{warning 'header is generated please add your documentation'}
METHOD testAnyStringIsEmpty : BOOL
VAR_INPUT
	inputStruct	: isEmptyDataStr;
	testNumber 	: USINT;
END_VAR

VAR
	message : STRING;
END_VAR
THIS^.reset();

IF (inputStruct.typeToTest = TypeToTest.TEST_WSTRING) THEN
	THIS^.assertorContainer.assertor.assert.strings.anyString.isEmpty(
		stringToCheck 	:= inputStruct.WStringToTest,
		message			:= ''
	);
					
ELSIF  (inputStruct.typeToTest = TypeToTest.TEST_STRING ) THEN
	THIS^.assertorContainer.assertor.assert.strings.anyString.isEmpty(
		stringToCheck 	:= inputStruct.StringToTest,
		message			:= ''
	);
	
END_IF

message	:= CONCAT( 'Test Number ', TO_STRING(testNumber));
message	:= CONCAT( message, ' during function AnyString.isEmpty ');
message	:= CONCAT( Message , ' has failed ');

THIS^.AssertEquals_BOOL(
	Expected 	:= inputStruct.expectedResult,
	Actual 		:= THIS^.assertorContainer.wasAssertionWrong,
	Message 	:= message
);
END_METHOD

(*

short summary
=============

.. <legal notes>

legal notes
=================
| SPDX-FileCopyrightText: © 2023 ekvip automation GmbH <info@ekvip.de>
| SPDX-License-Identifier: Apache-2.0
| For details check: Apache-2.0_

.. _Apache-2.0: https://www.apache.org/licenses/LICENSE-2.0

.. </legal notes>

parameters
==========

*)

{warning 'header is generated please add your documentation'}
METHOD testAnyStringIsEqualTo : BOOL
VAR_INPUT
	inputStruct	: isEqualToDataStr;
	testNumber 	: USINT;
END_VAR

VAR
	message : STRING;
END_VAR
THIS^.reset();

IF (inputStruct.typeToTest = TypeToTest.TEST_WSTRING) THEN
	THIS^.assertorContainer.assertor.assert.strings.anyString.isEqualTo(
		stringToCheck 	:= inputStruct.WStringToTest,
		expected		:= inputStruct.EqualToWString,
		ignoreCases     := inputStruct.IgnoreCases,
		message			:= ''	 	
	);
					
ELSIF  (inputStruct.typeToTest = TypeToTest.TEST_STRING ) THEN
	THIS^.assertorContainer.assertor.assert.strings.anyString.isEqualTo(
		stringToCheck 	:= inputStruct.StringToTest,
		expected		:= inputStruct.EqualToString,
		ignoreCases     := inputStruct.IgnoreCases,
		message			:= ''
	);
	
END_IF

message	:= CONCAT( 'Test Number ', TO_STRING(testNumber));
message	:= CONCAT( message, ' during function AnyString.isEqualTo ');
message	:= CONCAT( Message , ' has failed ');

THIS^.AssertEquals_BOOL(
	Expected 	:= inputStruct.expectedResult,
	Actual 		:= THIS^.assertorContainer.wasAssertionWrong,
	Message 	:= message
);
END_METHOD

(*

short summary
=============

.. <legal notes>

legal notes
=================
| SPDX-FileCopyrightText: © 2023 ekvip automation GmbH <info@ekvip.de>
| SPDX-License-Identifier: Apache-2.0
| For details check: Apache-2.0_

.. _Apache-2.0: https://www.apache.org/licenses/LICENSE-2.0

.. </legal notes>

parameters
==========

*)

{warning 'header is generated please add your documentation'}
METHOD testAnyStringIsNotEmpty : BOOL
VAR_INPUT
	inputStruct	: isEmptyDataStr;
	testNumber 	: USINT;
END_VAR

VAR
	message : STRING;
END_VAR
THIS^.reset();

IF (inputStruct.typeToTest = TypeToTest.TEST_WSTRING) THEN
	THIS^.assertorContainer.assertor.assert.strings.anyString.isNotEmpty(
		stringToCheck 	:= inputStruct.WStringToTest,
		message			:= ''
	);
					
ELSIF  (inputStruct.typeToTest = TypeToTest.TEST_STRING ) THEN
	THIS^.assertorContainer.assertor.assert.strings.anyString.isNotEmpty(
		stringToCheck 	:= inputStruct.StringToTest,
		message			:= ''
	);
	
END_IF

message	:= CONCAT( 'Test Number ', TO_STRING(testNumber));
message	:= CONCAT( message, ' during function AnyString.isNotEmpty ');
message	:= CONCAT( Message , ' has failed ');

THIS^.AssertEquals_BOOL(
	Expected 	:= inputStruct.expectedResult,
	Actual 		:= THIS^.assertorContainer.wasAssertionWrong,
	Message 	:= message
);
END_METHOD

(*

short summary
=============

.. <legal notes>

legal notes
=================
| SPDX-FileCopyrightText: © 2023 ekvip automation GmbH <info@ekvip.de>
| SPDX-License-Identifier: Apache-2.0
| For details check: Apache-2.0_

.. _Apache-2.0: https://www.apache.org/licenses/LICENSE-2.0

.. </legal notes>

parameters
==========

*)

{warning 'header is generated please add your documentation'}
METHOD testAnyStringIsNotEqualTo : BOOL
VAR_INPUT
	inputStruct	: isEqualToDataStr;
	testNumber 	: USINT;
END_VAR

VAR
	message : STRING;
END_VAR
THIS^.reset();

IF (inputStruct.typeToTest = TypeToTest.TEST_WSTRING) THEN
	THIS^.assertorContainer.assertor.assert.strings.anyString.isNotEqualTo(
		stringToCheck 	:= inputStruct.WStringToTest,
		unexpected		:= inputStruct.EqualToWString,
		ignoreCases     := inputStruct.IgnoreCases,
		message			:= ''	 	
	);
					
ELSIF  (inputStruct.typeToTest = TypeToTest.TEST_STRING ) THEN
	THIS^.assertorContainer.assertor.assert.strings.anyString.isNotEqualTo(
		stringToCheck 	:= inputStruct.StringToTest,
		unexpected		:= inputStruct.EqualToString,
		ignoreCases     := inputStruct.IgnoreCases,
		message			:= ''
	);
	
END_IF

message	:= CONCAT( 'Test Number ', TO_STRING(testNumber));
message	:= CONCAT( message, ' during function AnyString.isNotEqualTo ');
message	:= CONCAT( Message , ' has failed ');

THIS^.AssertEquals_BOOL(
	Expected 	:= inputStruct.expectedResult,
	Actual 		:= THIS^.assertorContainer.wasAssertionWrong,
	Message 	:= message
);
END_METHOD

(*

short summary
=============

.. <legal notes>

legal notes
=================
| SPDX-FileCopyrightText: © 2023 ekvip automation GmbH <info@ekvip.de>
| SPDX-License-Identifier: Apache-2.0
| For details check: Apache-2.0_

.. _Apache-2.0: https://www.apache.org/licenses/LICENSE-2.0

.. </legal notes>

parameters
==========

*)

{warning 'header is generated please add your documentation'}
METHOD testAnyStringLengthBetween
VAR_INPUT
	inputStruct	: IsLengthBetweenBasicData;
	testNumber	: USINT;
END_VAR

VAR
	message	: STRING;
END_VAR

THIS^.reset();

IF (inputStruct.typeToTest = TypeToTest.TEST_WSTRING) THEN	
	THIS^.assertorContainer.assertor.assert.strings.anyString.lenghtIsBetween( 
		stringToCheck	:=	inputStruct.wstringToTest, 
		maxLenght		:=	inputStruct.maxLength,
		minLenght   	:=  inputStruct.minLength,
		message			:=	''          
	);
				
ELSIF  (inputStruct.typeToTest = TypeToTest.TEST_STRING ) THEN
    THIS^.assertorContainer.assertor.assert.strings.anyString.lenghtIsBetween( 
		stringToCheck	:=	inputStruct.stringToTest, 
		maxLenght		:=	inputStruct.maxLength,
		minLenght   	:=  inputStruct.minLength,
		message			:=	''          
	);
END_IF

message	:= CONCAT( 'Test Number ', TO_STRING(testNumber));
message	:= CONCAT( message, ' during function AnyString.isLengthBetween ');
message	:= CONCAT( Message , ' has failed ');
	
THIS^.AssertEquals_BOOL(
	Expected 	:= inputStruct.expectedResult,
	Actual 		:= THIS^.assertorContainer.wasAssertionWrong,
	Message 	:= message
);
	
//TEST_FINISHED();
END_METHOD

(*

short summary
=============

.. <legal notes>

legal notes
=================
| SPDX-FileCopyrightText: © 2023 ekvip automation GmbH <info@ekvip.de>
| SPDX-License-Identifier: Apache-2.0
| For details check: Apache-2.0_

.. _Apache-2.0: https://www.apache.org/licenses/LICENSE-2.0

.. </legal notes>

parameters
==========

*)

{warning 'header is generated please add your documentation'}
METHOD testAnyStringLengthIs
VAR_INPUT
	inputStruct	:IsLengthBasicData;
	testNumber :USINT;
END_VAR

VAR
	message: STRING;
END_VAR


THIS^.reset();

IF (inputStruct.typeToTest = TypeToTest.TEST_WSTRING) THEN
	IF (inputStruct.funcType = FunctionType.EXACT) THEN 
		THIS^.assertorContainer.assertor.assert.strings.anyString.lenghtIsExact( 
			stringToCheck	:=	inputStruct.wstringToTest, 
			expectedLength	:=	inputStruct.expectedLength,
			message			:=	''          
		);
	ELSIF (inputStruct.funcType = FunctionType.MAXIMUM) THEN
		THIS^.assertorContainer.assertor.assert.strings.anyString.lenghtIsMax( 
			stringToCheck	:=	inputStruct.wstringToTest, 
			maxLength		:=	inputStruct.expectedLength,
			message			:=	''
		);
	ELSIF (inputStruct.funcType = FunctionType.MINIMUM) THEN
		THIS^.assertorContainer.assertor.assert.strings.anyString.lenghtIsMin( 
			stringToCheck	:=	inputStruct.wstringToTest, 
			minLength		:=	inputStruct.expectedLength,
			message			:=	''
		);
	END_IF;
				
ELSIF  (inputStruct.typeToTest = TypeToTest.TEST_STRING ) THEN
    IF (inputStruct.funcType = FunctionType.EXACT) THEN 
		THIS^.assertorContainer.assertor.assert.strings.anyString.lenghtIsExact( 
			stringToCheck	:=	inputStruct.stringToTest, 
			expectedLength	:=	inputStruct.expectedLength,
			message			:=	''         
		);
	ELSIF (inputStruct.funcType = FunctionType.MAXIMUM) THEN
		THIS^.assertorContainer.assertor.assert.strings.anyString.lenghtIsMax( 
			stringToCheck	:=	inputStruct.stringToTest, 
			maxLength		:=	inputStruct.expectedLength,
			message			:=	''        
		);
	ELSIF (inputStruct.funcType = FunctionType.MINIMUM) THEN
		THIS^.assertorContainer.assertor.assert.strings.anyString.lenghtIsMin( 
			stringToCheck	:=	inputStruct.stringToTest, 
			minLength		:=	inputStruct.expectedLength,
			message			:=	''          
		);
	END_IF;

END_IF

message	:= CONCAT( 'Test Number ', TO_STRING(testNumber));
message	:= CONCAT( message, ' during function AnyString.isLength ');
message	:= CONCAT( message , TO_STRING(inputStruct.funcType));
message	:= CONCAT( Message , ' has failed ');
	
THIS^.AssertEquals_BOOL(
	Expected 	:= inputStruct.expectedResult,
	Actual 		:= THIS^.assertorContainer.wasAssertionWrong,
	Message 	:= message
);
	
//TEST_FINISHED();
END_METHOD

(*

short summary
=============

.. <legal notes>

legal notes
=================
| SPDX-FileCopyrightText: © 2023 ekvip automation GmbH <info@ekvip.de>
| SPDX-License-Identifier: Apache-2.0
| For details check: Apache-2.0_

.. _Apache-2.0: https://www.apache.org/licenses/LICENSE-2.0

.. </legal notes>

parameters
==========

*)

{warning 'header is generated please add your documentation'}
METHOD testAnyStringStartsWith : BOOL
VAR_INPUT
	inputStruct	: containsDataStr;
	testNumber 	: USINT;
END_VAR

VAR
	message : STRING;
END_VAR
THIS^.reset();

IF (inputStruct.typeToTest = TypeToTest.TEST_WSTRING) THEN
	THIS^.assertorContainer.assertor.assert.strings.anyString.startsWith(
		stringToCheck	:= inputStruct.WStringToTest,
		start			:= inputStruct.WStringToContain,
		ignoreCases		:= inputStruct.IgnoreCases,
		trim			:= inputStruct.Trim,
		message			:= ''
	);
					
ELSIF  (inputStruct.typeToTest = TypeToTest.TEST_STRING ) THEN
	THIS^.assertorContainer.assertor.assert.strings.anyString.startsWith(
		stringToCheck	:= inputStruct.StringToTest,
		start			:= inputStruct.StringToContain,
		ignoreCases		:= inputStruct.IgnoreCases,
		trim			:= inputStruct.Trim,
		message			:= ''
	);

END_IF

message	:= CONCAT( 'Test Number ', TO_STRING(testNumber));
message	:= CONCAT( message, ' during function AnyString.startsWith ');
message	:= CONCAT( Message , ' has failed ');

THIS^.AssertEquals_BOOL(
	Expected 	:= inputStruct.expectedResult,
	Actual 		:= THIS^.assertorContainer.wasAssertionWrong,
	Message 	:= message
);
END_METHOD

(*

short summary
=============

.. <legal notes>

legal notes
=================
| SPDX-FileCopyrightText: © 2023 ekvip automation GmbH <info@ekvip.de>
| SPDX-License-Identifier: Apache-2.0
| For details check: Apache-2.0_

.. _Apache-2.0: https://www.apache.org/licenses/LICENSE-2.0

.. </legal notes>

parameters
==========

*)

{warning 'header is generated please add your documentation'}
METHOD testAsciiEndsWith : BOOL
VAR_INPUT
	inputStruct	: containsDataStr;
	testNumber 	: USINT;
END_VAR

VAR
	message : STRING;
END_VAR
THIS^.reset();

THIS^.assertorContainer.assertor.assert.strings.ascii.endsWith(
	stringToCheck	:= inputStruct.StringToTest,
	end				:= inputStruct.StringToContain,
	ignoreCases		:= inputStruct.IgnoreCases,
	trim			:= inputStruct.Trim,
	message			:= ''
);


message	:= CONCAT( 'Test Number ', TO_STRING(testNumber));
message	:= CONCAT( message, ' during function Ascii.endsWith ');
message	:= CONCAT( Message , ' has failed ');

THIS^.AssertEquals_BOOL(
	Expected 	:= inputStruct.expectedResult,
	Actual 		:= THIS^.assertorContainer.wasAssertionWrong,
	Message 	:= message
);
END_METHOD

(*

short summary
=============

.. <legal notes>

legal notes
=================
| SPDX-FileCopyrightText: © 2023 ekvip automation GmbH <info@ekvip.de>
| SPDX-License-Identifier: Apache-2.0
| For details check: Apache-2.0_

.. _Apache-2.0: https://www.apache.org/licenses/LICENSE-2.0

.. </legal notes>

parameters
==========

*)

{warning 'header is generated please add your documentation'}
METHOD testAsciiIsEmpty : BOOL
VAR_INPUT
	inputStruct	: isEmptyDataStr;
	testNumber 	: USINT;
END_VAR

VAR
	message : STRING;
END_VAR
THIS^.reset();

THIS^.assertorContainer.assertor.assert.strings.anyString.isEmpty(
	stringToCheck 	:= inputStruct.StringToTest,
	message			:= ''
);

message	:= CONCAT( 'Test Number ', TO_STRING(testNumber));
message	:= CONCAT( message, ' during function Ascii.isEmpty ');
message	:= CONCAT( Message , ' has failed ');

THIS^.AssertEquals_BOOL(
	Expected 	:= inputStruct.expectedResult,
	Actual 		:= THIS^.assertorContainer.wasAssertionWrong,
	Message 	:= message
);
END_METHOD

(*

short summary
=============

.. <legal notes>

legal notes
=================
| SPDX-FileCopyrightText: © 2023 ekvip automation GmbH <info@ekvip.de>
| SPDX-License-Identifier: Apache-2.0
| For details check: Apache-2.0_

.. _Apache-2.0: https://www.apache.org/licenses/LICENSE-2.0

.. </legal notes>

parameters
==========

*)

{warning 'header is generated please add your documentation'}
METHOD testAsciiIsEqualTo : BOOL
VAR_INPUT
	inputStruct	: isEqualToDataStr;
	testNumber 	: USINT;
END_VAR

VAR
	message : STRING;
END_VAR
THIS^.reset();

THIS^.assertorContainer.assertor.assert.strings.ascii.isEqualTo(
	stringToCheck 	:= inputStruct.StringToTest,
	expected		:= inputStruct.EqualToString,
	ignoreCases     := inputStruct.IgnoreCases,
	message			:= ''	 	
);

message	:= CONCAT( 'Test Number ', TO_STRING(testNumber));
message	:= CONCAT( message, ' during function Ascii.isEqualTo ');
message	:= CONCAT( Message , ' has failed ');

THIS^.AssertEquals_BOOL(
	Expected 	:= inputStruct.expectedResult,
	Actual 		:= THIS^.assertorContainer.wasAssertionWrong,
	Message 	:= message
);
END_METHOD

(*

short summary
=============

.. <legal notes>

legal notes
=================
| SPDX-FileCopyrightText: © 2023 ekvip automation GmbH <info@ekvip.de>
| SPDX-License-Identifier: Apache-2.0
| For details check: Apache-2.0_

.. _Apache-2.0: https://www.apache.org/licenses/LICENSE-2.0

.. </legal notes>

parameters
==========

*)

{warning 'header is generated please add your documentation'}
METHOD testAsciiIsNotEmpty : BOOL
VAR_INPUT
	inputStruct	: isEmptyDataStr;
	testNumber 	: USINT;
END_VAR

VAR
	message : STRING;
END_VAR
THIS^.reset();

THIS^.assertorContainer.assertor.assert.strings.anyString.isNotEmpty(
	stringToCheck 	:= inputStruct.StringToTest,
	message			:= ''
);

message	:= CONCAT( 'Test Number ', TO_STRING(testNumber));
message	:= CONCAT( message, ' during function Ascii.isNotEmpty ');
message	:= CONCAT( Message , ' has failed ');

THIS^.AssertEquals_BOOL(
	Expected 	:= inputStruct.expectedResult,
	Actual 		:= THIS^.assertorContainer.wasAssertionWrong,
	Message 	:= message
);
END_METHOD

(*

short summary
=============

.. <legal notes>

legal notes
=================
| SPDX-FileCopyrightText: © 2023 ekvip automation GmbH <info@ekvip.de>
| SPDX-License-Identifier: Apache-2.0
| For details check: Apache-2.0_

.. _Apache-2.0: https://www.apache.org/licenses/LICENSE-2.0

.. </legal notes>

parameters
==========

*)

{warning 'header is generated please add your documentation'}
METHOD testAsciiIsNotEqualTo : BOOL
VAR_INPUT
	inputStruct	: isEqualToDataStr;
	testNumber 	: USINT;
END_VAR

VAR
	message : STRING;
END_VAR
THIS^.reset();

THIS^.assertorContainer.assertor.assert.strings.anyString.isNotEqualTo(
	stringToCheck 	:= inputStruct.StringToTest,
	unexpected		:= inputStruct.EqualToString,
	ignoreCases     := inputStruct.IgnoreCases,
	message			:= ''	 	
);

message	:= CONCAT( 'Test Number ', TO_STRING(testNumber));
message	:= CONCAT( message, ' during function Ascii.isNotEqualTo ');
message	:= CONCAT( Message , ' has failed ');

THIS^.AssertEquals_BOOL(
	Expected 	:= inputStruct.expectedResult,
	Actual 		:= THIS^.assertorContainer.wasAssertionWrong,
	Message 	:= message
);
END_METHOD

(*

short summary
=============

.. <legal notes>

legal notes
=================
| SPDX-FileCopyrightText: © 2023 ekvip automation GmbH <info@ekvip.de>
| SPDX-License-Identifier: Apache-2.0
| For details check: Apache-2.0_

.. _Apache-2.0: https://www.apache.org/licenses/LICENSE-2.0

.. </legal notes>

parameters
==========

*)

{warning 'header is generated please add your documentation'}
METHOD testAsciiStartsWith : BOOL
VAR_INPUT
	inputStruct	: containsDataStr;
	testNumber 	: USINT;
END_VAR

VAR
	message : STRING;
END_VAR
THIS^.reset();

THIS^.assertorContainer.assertor.assert.strings.ascii.startsWith(
	stringToCheck	:= inputStruct.StringToTest,
	start			:= inputStruct.StringToContain,
	ignoreCases		:= inputStruct.IgnoreCases,
	trim			:= inputStruct.Trim,
	message			:= ''
);


message	:= CONCAT( 'Test Number ', TO_STRING(testNumber));
message	:= CONCAT( message, ' during function Ascii.startsWith ');
message	:= CONCAT( Message , ' has failed ');

THIS^.AssertEquals_BOOL(
	Expected 	:= inputStruct.expectedResult,
	Actual 		:= THIS^.assertorContainer.wasAssertionWrong,
	Message 	:= message
);
END_METHOD

(*

short summary
=============

.. <legal notes>

legal notes
=================
| SPDX-FileCopyrightText: © 2023 ekvip automation GmbH <info@ekvip.de>
| SPDX-License-Identifier: Apache-2.0
| For details check: Apache-2.0_

.. _Apache-2.0: https://www.apache.org/licenses/LICENSE-2.0

.. </legal notes>

parameters
==========

*)

{warning 'header is generated please add your documentation'}
METHOD testAsciiStringContains : BOOL
VAR_INPUT
	inputStruct	: containsDataStr;
	testNumber :USINT;
END_VAR

VAR
	message : STRING;
END_VAR
THIS^.reset();

THIS^.assertorContainer.assertor.assert.strings.ascii.contains(
	stringToCheck 	:= inputStruct.StringToTest,
	searchString	:= inputStruct.StringToContain, 
	ignoreCases		:= inputStruct.IgnoreCases,
	message         := ''
);

message	:= CONCAT( 'Test Number ', TO_STRING(testNumber));
message	:= CONCAT( message, ' during function Ascii.contains ');
message	:= CONCAT( Message , ' has failed ');

THIS^.AssertEquals_BOOL(
	Expected 	:= inputStruct.expectedResult,
	Actual 		:= THIS^.assertorContainer.wasAssertionWrong,
	Message 	:= message
);
END_METHOD

(*

short summary
=============

.. <legal notes>

legal notes
=================
| SPDX-FileCopyrightText: © 2023 ekvip automation GmbH <info@ekvip.de>
| SPDX-License-Identifier: Apache-2.0
| For details check: Apache-2.0_

.. _Apache-2.0: https://www.apache.org/licenses/LICENSE-2.0

.. </legal notes>

parameters
==========

*)

{warning 'header is generated please add your documentation'}
METHOD testAsciiStringContainsNo : BOOL
VAR_INPUT
	inputStruct	: containsDataStr;
	testNumber 	: USINT;
END_VAR

VAR
	message : STRING;
END_VAR
THIS^.reset();

THIS^.assertorContainer.assertor.assert.strings.utf16.containsNo(
	stringToCheck 	:= inputStruct.WStringToTest,
	searchString	:= inputStruct.WStringToContain, 
	ignoreCases		:= inputStruct.IgnoreCases,
	message         := ''
);

message	:= CONCAT( 'Test Number ', TO_STRING(testNumber));
message	:= CONCAT( message, ' during function Ascii.containsNo ');
message	:= CONCAT( Message , ' has failed ');

THIS^.AssertEquals_BOOL(
	Expected 	:= inputStruct.expectedResult,
	Actual 		:= THIS^.assertorContainer.wasAssertionWrong,
	Message 	:= message
);
END_METHOD

(*

short summary
=============

.. <legal notes>

legal notes
=================
| SPDX-FileCopyrightText: © 2023 ekvip automation GmbH <info@ekvip.de>
| SPDX-License-Identifier: Apache-2.0
| For details check: Apache-2.0_

.. _Apache-2.0: https://www.apache.org/licenses/LICENSE-2.0

.. </legal notes>

parameters
==========

*)

{warning 'header is generated please add your documentation'}
METHOD testAsciiStringLengthBetween
VAR_INPUT
	inputStruct	: IsLengthBetweenBasicData;
	testNumber 	: USINT;
END_VAR

VAR
	message : STRING;
END_VAR
THIS^.reset();

THIS^.assertorContainer.assertor.assert.strings.ascii.lenghtIsBetween( 
	stringToCheck	:=	inputStruct.stringToTest, 
	maxLenght		:=	inputStruct.maxLength,
	minLenght   	:=  inputStruct.minLength,
	message			:=	''          
);


message	:= CONCAT( 'Test Number ', TO_STRING(testNumber));
message	:= CONCAT( message, ' during function Ascii.isLengthBetween ');
message	:= CONCAT( Message , ' has failed ');
	
THIS^.AssertEquals_BOOL(
	Expected 	:= inputStruct.expectedResult,
	Actual 		:= THIS^.assertorContainer.wasAssertionWrong,
	Message 	:= message
);
END_METHOD

(*

short summary
=============

.. <legal notes>

legal notes
=================
| SPDX-FileCopyrightText: © 2023 ekvip automation GmbH <info@ekvip.de>
| SPDX-License-Identifier: Apache-2.0
| For details check: Apache-2.0_

.. _Apache-2.0: https://www.apache.org/licenses/LICENSE-2.0

.. </legal notes>

parameters
==========

*)

{warning 'header is generated please add your documentation'}
METHOD testAsciiStringlengthIs
VAR_INPUT
	inputStruct	:IsLengthBasicData;
	testNumber :USINT;
END_VAR

VAR
	message: STRING;
END_VAR

THIS^.reset();

IF (inputStruct.funcType = FunctionType.EXACT) THEN 
	THIS^.assertorContainer.assertor.assert.strings.ascii.lenghtIsExact( 
		stringToCheck	:=	inputStruct.stringToTest, 
		expectedLength	:=	TO_USINT(inputStruct.expectedLength),
		message			:=	''          
	);
ELSIF (inputStruct.funcType = FunctionType.MAXIMUM) THEN
	THIS^.assertorContainer.assertor.assert.strings.ascii.lenghtIsMax( 
		stringToCheck	:=	inputStruct.stringToTest, 
		maxLength		:=	TO_USINT(inputStruct.expectedLength),
		message			:=	''         
	);
ELSIF (inputStruct.funcType = FunctionType.MINIMUM) THEN
	THIS^.assertorContainer.assertor.assert.strings.ascii.lenghtIsMin( 
		stringToCheck	:=	inputStruct.stringToTest, 
		minLength		:=	TO_USINT(inputStruct.expectedLength),
		message			:=	''          
	);
END_IF;

message	:= CONCAT( 'Test Number ', TO_STRING(testNumber));
message	:= CONCAT( message, ' during function AsciiString.isLength ');
message	:= CONCAT( message , TO_STRING(inputStruct.funcType));
message	:= CONCAT( Message , ' has failed ');

THIS^.AssertEquals_BOOL(
	Expected 	:= inputStruct.expectedResult,
	Actual 		:= THIS^.assertorContainer.wasAssertionWrong,
	Message		:= message
);
END_METHOD

(*

short summary
=============

.. <legal notes>

legal notes
=================
| SPDX-FileCopyrightText: © 2023 ekvip automation GmbH <info@ekvip.de>
| SPDX-License-Identifier: Apache-2.0
| For details check: Apache-2.0_

.. _Apache-2.0: https://www.apache.org/licenses/LICENSE-2.0

.. </legal notes>

parameters
==========

*)

{warning 'header is generated please add your documentation'}
METHOD testUtf16EndsWith : BOOL
VAR_INPUT
	inputStruct	: containsDataStr;
	testNumber 	: USINT;
END_VAR

VAR
	message : STRING;
END_VAR
THIS^.reset();

THIS^.assertorContainer.assertor.assert.strings.utf16.endsWith(
	stringToCheck	:= inputStruct.WStringToTest,
	end				:= inputStruct.WStringToContain,
	ignoreCases		:= inputStruct.IgnoreCases,
	trim			:= inputStruct.Trim,
	message			:= ''
);

message	:= CONCAT( 'Test Number ', TO_STRING(testNumber));
message	:= CONCAT( message, ' during function UTF16.endsWith ');
message	:= CONCAT( Message , ' has failed ');

THIS^.AssertEquals_BOOL(
	Expected 	:= inputStruct.expectedResult,
	Actual 		:= THIS^.assertorContainer.wasAssertionWrong,
	Message 	:= message
);
END_METHOD

(*

short summary
=============

.. <legal notes>

legal notes
=================
| SPDX-FileCopyrightText: © 2023 ekvip automation GmbH <info@ekvip.de>
| SPDX-License-Identifier: Apache-2.0
| For details check: Apache-2.0_

.. _Apache-2.0: https://www.apache.org/licenses/LICENSE-2.0

.. </legal notes>

parameters
==========

*)

{warning 'header is generated please add your documentation'}
METHOD testUtf16IsEmpty : BOOL
VAR_INPUT
	inputStruct	: isEmptyDataStr;
	testNumber 	: USINT;
END_VAR

VAR
	message : STRING;
END_VAR
THIS^.reset();

THIS^.assertorContainer.assertor.assert.strings.anyString.isEmpty(
	stringToCheck 	:= inputStruct.WStringToTest,
	message			:= ''
);

message	:= CONCAT( 'Test Number ', TO_STRING(testNumber));
message	:= CONCAT( message, ' during function UTF16.isEmpty ');
message	:= CONCAT( Message , ' has failed ');

THIS^.AssertEquals_BOOL(
	Expected 	:= inputStruct.expectedResult,
	Actual 		:= THIS^.assertorContainer.wasAssertionWrong,
	Message 	:= message
);
END_METHOD

(*

short summary
=============

.. <legal notes>

legal notes
=================
| SPDX-FileCopyrightText: © 2023 ekvip automation GmbH <info@ekvip.de>
| SPDX-License-Identifier: Apache-2.0
| For details check: Apache-2.0_

.. _Apache-2.0: https://www.apache.org/licenses/LICENSE-2.0

.. </legal notes>

parameters
==========

*)

{warning 'header is generated please add your documentation'}
METHOD testUtf16IsEqualTo : BOOL
VAR_INPUT
	inputStruct	: isEqualToDataStr;
	testNumber 	: USINT;
END_VAR

VAR
	message : STRING;
END_VAR
THIS^.reset();

THIS^.assertorContainer.assertor.assert.strings.anyString.isEqualTo(
	stringToCheck 	:= inputStruct.WStringToTest,
	expected		:= inputStruct.EqualToWString,
	ignoreCases     := inputStruct.IgnoreCases,
	message			:= ''	 	
);
   
message	:= CONCAT( 'Test Number ', TO_STRING(testNumber));
message	:= CONCAT( message, ' during function UTF16.isEqualTo ');
message	:= CONCAT( Message , ' has failed ');

THIS^.AssertEquals_BOOL(
	Expected 	:= inputStruct.expectedResult,
	Actual 		:= THIS^.assertorContainer.wasAssertionWrong,
	Message 	:= message
);
END_METHOD

(*

short summary
=============

.. <legal notes>

legal notes
=================
| SPDX-FileCopyrightText: © 2023 ekvip automation GmbH <info@ekvip.de>
| SPDX-License-Identifier: Apache-2.0
| For details check: Apache-2.0_

.. _Apache-2.0: https://www.apache.org/licenses/LICENSE-2.0

.. </legal notes>

parameters
==========

*)

{warning 'header is generated please add your documentation'}
METHOD testUtf16IsNotEmpty : BOOL
VAR_INPUT
	inputStruct	: isEmptyDataStr;
	testNumber 	: USINT;
END_VAR

VAR
	message : STRING;
END_VAR
THIS^.reset();

THIS^.assertorContainer.assertor.assert.strings.anyString.isNotEmpty(
	stringToCheck 	:= inputStruct.WStringToTest,
	message			:= ''
);

message	:= CONCAT( 'Test Number ', TO_STRING(testNumber));
message	:= CONCAT( message, ' during function UTF16.isNotEmpty ');
message	:= CONCAT( Message , ' has failed ');

THIS^.AssertEquals_BOOL(
	Expected 	:= inputStruct.expectedResult,
	Actual 		:= THIS^.assertorContainer.wasAssertionWrong,
	Message 	:= message
);
END_METHOD

(*

short summary
=============

.. <legal notes>

legal notes
=================
| SPDX-FileCopyrightText: © 2023 ekvip automation GmbH <info@ekvip.de>
| SPDX-License-Identifier: Apache-2.0
| For details check: Apache-2.0_

.. _Apache-2.0: https://www.apache.org/licenses/LICENSE-2.0

.. </legal notes>

parameters
==========

*)

{warning 'header is generated please add your documentation'}
METHOD testUtf16IsNotEqualTo : BOOL
VAR_INPUT
	inputStruct	: isEqualToDataStr;
	testNumber 	: USINT;
END_VAR

VAR
	message : STRING;
END_VAR
THIS^.reset();

THIS^.assertorContainer.assertor.assert.strings.anyString.isNotEqualTo(
	stringToCheck 	:= inputStruct.WStringToTest,
	unexpected		:= inputStruct.EqualToWString,
	ignoreCases     := inputStruct.IgnoreCases,
	message			:= ''	 	
);
   
message	:= CONCAT( 'Test Number ', TO_STRING(testNumber));
message	:= CONCAT( message, ' during function UTF16.isNotEqualTo ');
message	:= CONCAT( Message , ' has failed ');

THIS^.AssertEquals_BOOL(
	Expected 	:= inputStruct.expectedResult,
	Actual 		:= THIS^.assertorContainer.wasAssertionWrong,
	Message 	:= message
);
END_METHOD

(*

short summary
=============

.. <legal notes>

legal notes
=================
| SPDX-FileCopyrightText: © 2023 ekvip automation GmbH <info@ekvip.de>
| SPDX-License-Identifier: Apache-2.0
| For details check: Apache-2.0_

.. _Apache-2.0: https://www.apache.org/licenses/LICENSE-2.0

.. </legal notes>

parameters
==========

*)

{warning 'header is generated please add your documentation'}
METHOD testUtf16StartsWith : BOOL
VAR_INPUT
	inputStruct	: containsDataStr;
	testNumber 	: USINT;
END_VAR

VAR
	message : STRING;
END_VAR
THIS^.reset();

THIS^.assertorContainer.assertor.assert.strings.utf16.startsWith(
	stringToCheck	:= inputStruct.WStringToTest,
	start			:= inputStruct.WStringToContain,
	ignoreCases		:= inputStruct.IgnoreCases,
	trim			:= inputStruct.Trim,
	message			:= ''
);

message	:= CONCAT( 'Test Number ', TO_STRING(testNumber));
message	:= CONCAT( message, ' during function UTF16.startsWith ');
message	:= CONCAT( Message , ' has failed ');

THIS^.AssertEquals_BOOL(
	Expected 	:= inputStruct.expectedResult,
	Actual 		:= THIS^.assertorContainer.wasAssertionWrong,
	Message 	:= message
);
END_METHOD

(*

short summary
=============

.. <legal notes>

legal notes
=================
| SPDX-FileCopyrightText: © 2023 ekvip automation GmbH <info@ekvip.de>
| SPDX-License-Identifier: Apache-2.0
| For details check: Apache-2.0_

.. _Apache-2.0: https://www.apache.org/licenses/LICENSE-2.0

.. </legal notes>

parameters
==========

*)

{warning 'header is generated please add your documentation'}
METHOD testUtf16StringContains : BOOL
VAR_INPUT
	inputStruct	: containsDataStr;
	testNumber :USINT;
END_VAR

VAR
	message : STRING;
END_VAR
THIS^.reset();

THIS^.assertorContainer.assertor.assert.strings.utf16.contains(
	stringToCheck 	:= inputStruct.WStringToTest,
	searchString	:= inputStruct.WStringToContain, 
	ignoreCases		:= inputStruct.IgnoreCases,
	message         := ''
);

message	:= CONCAT( 'Test Number ', TO_STRING(testNumber));
message	:= CONCAT( message, ' during function UTF16.contains ');
message	:= CONCAT( Message , ' has failed ');

THIS^.AssertEquals_BOOL(
	Expected 	:= inputStruct.expectedResult,
	Actual 		:= THIS^.assertorContainer.wasAssertionWrong,
	Message 	:= message
);
END_METHOD

(*

short summary
=============

.. <legal notes>

legal notes
=================
| SPDX-FileCopyrightText: © 2023 ekvip automation GmbH <info@ekvip.de>
| SPDX-License-Identifier: Apache-2.0
| For details check: Apache-2.0_

.. _Apache-2.0: https://www.apache.org/licenses/LICENSE-2.0

.. </legal notes>

parameters
==========

*)

{warning 'header is generated please add your documentation'}
METHOD testUtf16StringContainsNo : BOOL
VAR_INPUT
	inputStruct	: containsDataStr;
	testNumber 	: USINT;
END_VAR

VAR
	message : STRING;
END_VAR
THIS^.reset();

THIS^.assertorContainer.assertor.assert.strings.utf16.containsNo(
	stringToCheck 	:= inputStruct.WStringToTest,
	searchString	:= inputStruct.WStringToContain, 
	ignoreCases		:= inputStruct.IgnoreCases,
	message         := ''
);

message	:= CONCAT( 'Test Number ', TO_STRING(testNumber));
message	:= CONCAT( message, ' during function UTF16.containsNo ');
message	:= CONCAT( Message , ' has failed ');

THIS^.AssertEquals_BOOL(
	Expected 	:= inputStruct.expectedResult,
	Actual 		:= THIS^.assertorContainer.wasAssertionWrong,
	Message 	:= message
);
END_METHOD

(*

short summary
=============

.. <legal notes>

legal notes
=================
| SPDX-FileCopyrightText: © 2023 ekvip automation GmbH <info@ekvip.de>
| SPDX-License-Identifier: Apache-2.0
| For details check: Apache-2.0_

.. _Apache-2.0: https://www.apache.org/licenses/LICENSE-2.0

.. </legal notes>

parameters
==========

*)

{warning 'header is generated please add your documentation'}
METHOD testUtf16StringLengthBetween
VAR_INPUT
	inputStruct : IsLengthBetweenBasicData;
	testNumber	: USINT;
END_VAR

VAR
	message: STRING;
END_VAR
THIS^.reset();

THIS^.assertorContainer.assertor.assert.strings.utf16.lenghtIsBetween( 
	stringToCheck	:=	inputStruct.wstringToTest, 
	maxLenght		:=	inputStruct.maxLength,
	minLenght   	:=  inputStruct.minLength,
	message			:=	''          
);


message	:= CONCAT( 'Test Number ', TO_STRING(testNumber));
message	:= CONCAT( message, ' during function UTF16.isLengthBetween ');
message	:= CONCAT( Message , ' has failed ');
	
THIS^.AssertEquals_BOOL(
	Expected 	:= inputStruct.expectedResult,
	Actual 		:= THIS^.assertorContainer.wasAssertionWrong,
	Message 	:= message
);
END_METHOD

(*

short summary
=============

.. <legal notes>

legal notes
=================
| SPDX-FileCopyrightText: © 2023 ekvip automation GmbH <info@ekvip.de>
| SPDX-License-Identifier: Apache-2.0
| For details check: Apache-2.0_

.. _Apache-2.0: https://www.apache.org/licenses/LICENSE-2.0

.. </legal notes>

parameters
==========

*)

{warning 'header is generated please add your documentation'}
METHOD testUtf16StringlengthIs
VAR_INPUT
	inputStruct	:IsLengthBasicData;
	testNumber :USINT;
END_VAR

VAR
	message: STRING;
END_VAR

THIS^.reset();

IF (inputStruct.funcType = FunctionType.EXACT) THEN
	THIS^.assertorContainer.assertor.assert.strings.utf16.lenghtIsExact( 
		stringToCheck	:=	inputStruct.wstringToTest, 
		expectedLength	:=	TO_USINT(inputStruct.expectedLength),
		message			:=	''          
	);
ELSIF (inputStruct.funcType = FunctionType.MAXIMUM) THEN
	THIS^.assertorContainer.assertor.assert.strings.utf16.lenghtIsMax( 
		stringToCheck	:=	inputStruct.wstringToTest, 
		maxLength		:=	TO_USINT(inputStruct.expectedLength),
		message			:=	''         
	);
ELSIF (inputStruct.funcType = FunctionType.MINIMUM) THEN
	THIS^.assertorContainer.assertor.assert.strings.utf16.lenghtIsMin( 
		stringToCheck	:=	inputStruct.wstringToTest, 
		minLength		:=	TO_USINT(inputStruct.expectedLength),
		message			:=	' '         
	);
END_IF;

message	:= CONCAT( ' Test Number ', TO_STRING(testNumber));
message	:= CONCAT( message, ' during function UFT16String.isLength ');
message	:= CONCAT( message , TO_STRING(inputStruct.funcType));
message	:= CONCAT( Message , ' has failed ');
	
THIS^.AssertEquals_BOOL(
	Expected 	:= inputStruct.expectedResult,
	Actual 		:= THIS^.assertorContainer.wasAssertionWrong,
	Message 	:= message
);
END_METHOD

END_FUNCTION_BLOCK

// ---- AssertionTester/AssertionTests/TimeAssertions/TimeAssertionsTests.TcPOU
(*

short summary
=============

.. <legal notes>

legal notes
=================
| SPDX-FileCopyrightText: © 2023 ekvip automation GmbH <info@ekvip.de>
| SPDX-License-Identifier: Apache-2.0
| For details check: Apache-2.0_

.. _Apache-2.0: https://www.apache.org/licenses/LICENSE-2.0

.. </legal notes>

methods and properties
======================

*)

{warning 'header is generated please add your documentation'}
FUNCTION_BLOCK TimeAssertionsTests EXTENDS AbstractAssertorTest
VAR CONSTANT
	NUMBER_OF_SETS :INT := 9;
END_VAR
VAR
	simpleTimeValuesToCurrent 	:ARRAY [0..NUMBER_OF_SETS] OF TIME;
	simpleTimeValuesToExpected 	:ARRAY [0..NUMBER_OF_SETS] OF TIME;
	longTimeValuesToCurrent 	:ARRAY [0..NUMBER_OF_SETS] OF LTIME;
	longTimeValuesToExpected 	:ARRAY [0..NUMBER_OF_SETS] OF LTIME;								
END_VAR


assignTimes();

(* Simple time tests *)

THIS^.testSimpleValueIsEqualTo(simpleTimeValuesToCurrent, simpleTimeValuesToExpected);

THIS^.testSimpleValueIsNotEqualTo(simpleTimeValuesToCurrent, mirrorSimpleTimeArray(simpleTimeValuesToExpected));

THIS^.testSimpleValueIsGreaterThan(simpleTimeValuesToCurrent, simpleTimeValuesToExpected);

THIS^.testSimpleValueIsLessThan(simpleTimeValuesToCurrent, simpleTimeValuesToExpected);

THIS^.testSimpleValueIsInRangeOf(simpleTimeValuesToCurrent, simpleTimeValuesToExpected, mirrorSimpleTimeArray(simpleTimeValuesToExpected));

THIS^.testSimpleValueIsMax(simpleTimeValuesToCurrent, mirrorSimpleTimeArray(simpleTimeValuesToExpected));

THIS^.testSimpleValueIsMin(simpleTimeValuesToCurrent, mirrorSimpleTimeArray(simpleTimeValuesToExpected));

THIS^.testSimpleTimeHasExpired(simpleTimeValuesToCurrent, mirrorSimpleTimeArray(simpleTimeValuesToExpected));

THIS^.testSimpleTimeHasNotExpired(simpleTimeValuesToCurrent, mirrorSimpleTimeArray(simpleTimeValuesToExpected));

(* Long time tests *)

THIS^.testLongValueIsEqualTo(longTimeValuesToCurrent, longTimeValuesToExpected);

THIS^.testLongValueIsNotEqualTo(longTimeValuesToCurrent, mirrorLongTimeArray(longTimeValuesToExpected));

THIS^.testLongValueIsGreaterThan(longTimeValuesToCurrent, longTimeValuesToExpected);

THIS^.testLongValueIsLessThan(longTimeValuesToCurrent, longTimeValuesToExpected);

THIS^.testLongValueIsInRangeOf(longTimeValuesToCurrent, longTimeValuesToExpected, mirrorLongTimeArray(longTimeValuesToExpected));

THIS^.testLongValueIsMax(longTimeValuesToCurrent, mirrorLongTimeArray(longTimeValuesToExpected));

THIS^.testLongValueIsMin(longTimeValuesToCurrent, mirrorLongTimeArray(longTimeValuesToExpected));

THIS^.testLongTimeHasExpired(longTimeValuesToCurrent, mirrorlongTimeArray(longTimeValuesToExpected));

THIS^.testLongTimeHasNotExpired(longTimeValuesToCurrent, mirrorlongTimeArray(longTimeValuesToExpected));

(*

short summary
=============

.. <legal notes>

legal notes
=================
| SPDX-FileCopyrightText: © 2023 ekvip automation GmbH <info@ekvip.de>
| SPDX-License-Identifier: Apache-2.0
| For details check: Apache-2.0_

.. _Apache-2.0: https://www.apache.org/licenses/LICENSE-2.0

.. </legal notes>

parameters
==========

*)

{warning 'header is generated please add your documentation'}
METHOD assignTimes
		
// simple time
simpleTimeValuesToCurrent[0] := TIME#0M;					simpleTimeValuesToExpected[0] := TIME#0S;
simpleTimeValuesToCurrent[1] := TIME#0.01667M;				simpleTimeValuesToExpected[1] := TIME#1S;
simpleTimeValuesToCurrent[2] := TIME#1M;					simpleTimeValuesToExpected[2] := TIME#60S;
simpleTimeValuesToCurrent[3] := TIME#60M;					simpleTimeValuesToExpected[3] := TIME#3_600S;
simpleTimeValuesToCurrent[4] := TIME#1440M;					simpleTimeValuesToExpected[4] := TIME#86_400S;
simpleTimeValuesToCurrent[5] := TIME#10_080M;				simpleTimeValuesToExpected[5] := TIME#604_800S;
simpleTimeValuesToCurrent[6] := TIME#20_160M;				simpleTimeValuesToExpected[6] := TIME#1_209_600S;
simpleTimeValuesToCurrent[7] := TIME#40_320M;				simpleTimeValuesToExpected[7] := TIME#2_419_200S;
simpleTimeValuesToCurrent[8] := TIME#60_480M;				simpleTimeValuesToExpected[8] := TIME#3_628_800S;
simpleTimeValuesToCurrent[9] := TIME#4294967295MS;			simpleTimeValuesToExpected[9] := TIME#4294967295MS;

// long time
longTimeValuesToCurrent[0] := LTIME#0MS;					longTimeValuesToExpected[0] := LTIME#0NS;
longTimeValuesToCurrent[1] := LTIME#1_000MS;				longTimeValuesToExpected[1] := LTIME#1000_000_000NS;
longTimeValuesToCurrent[2] := LTIME#60_000MS;				longTimeValuesToExpected[2] := LTIME#60_000_000_000NS;
longTimeValuesToCurrent[3] := LTIME#3_600_000MS;			longTimeValuesToExpected[3] := LTIME#3_600_000_000_000NS;
longTimeValuesToCurrent[4] := LTIME#86_400_000MS;			longTimeValuesToExpected[4] := LTIME#86_400_000_000_000NS;
longTimeValuesToCurrent[5] := LTIME#604_800_000MS;			longTimeValuesToExpected[5] := LTIME#604_800_000_000_000NS;
longTimeValuesToCurrent[6] := LTIME#1_209_600_000MS;		longTimeValuesToExpected[6] := LTIME#1_209_600_000_000_000NS;
longTimeValuesToCurrent[7] := LTIME#2_419_200_000MS;		longTimeValuesToExpected[7] := LTIME#2_419_200_000_000_000NS;
longTimeValuesToCurrent[8] := LTIME#31_557_600_000MS;		longTimeValuesToExpected[8] := LTIME#31_557_600_000_000_000NS;
longTimeValuesToCurrent[9] := LTIME#31_557_600_000MS;		longTimeValuesToExpected[9] := LTIME#213503D23H34M33S709MS551US615NS;
END_METHOD

(*

short summary
=============

.. <legal notes>

legal notes
=================
| SPDX-FileCopyrightText: © 2023 ekvip automation GmbH <info@ekvip.de>
| SPDX-License-Identifier: Apache-2.0
| For details check: Apache-2.0_

.. _Apache-2.0: https://www.apache.org/licenses/LICENSE-2.0

.. </legal notes>

parameters
==========

*)

{warning 'header is generated please add your documentation'}

METHOD mirrorLongTimeArray :ARRAY [0..NUMBER_OF_SETS] OF LTIME
VAR_INPUT
	inputArray :ARRAY [0..NUMBER_OF_SETS] OF LTIME;
END_VAR
VAR
	tempArray :ARRAY [0..NUMBER_OF_SETS] OF LTIME;
	temp :LTIME;
	i :INT;
END_VAR
tempArray := inputArray;

FOR i := 0 TO (NUMBER_OF_SETS/2 - 1) DO
	temp := inputArray[i];
	tempArray[i] := inputArray[NUMBER_OF_SETS - i];
	tempArray[NUMBER_OF_SETS - i] := temp;
END_FOR

mirrorLongTimeArray := tempArray;
END_METHOD

(*

short summary
=============

.. <legal notes>

legal notes
=================
| SPDX-FileCopyrightText: © 2023 ekvip automation GmbH <info@ekvip.de>
| SPDX-License-Identifier: Apache-2.0
| For details check: Apache-2.0_

.. _Apache-2.0: https://www.apache.org/licenses/LICENSE-2.0

.. </legal notes>

parameters
==========

*)

{warning 'header is generated please add your documentation'}

METHOD mirrorSimpleTimeArray :ARRAY [0..NUMBER_OF_SETS] OF TIME
VAR_INPUT
	inputArray :ARRAY [0..NUMBER_OF_SETS] OF TIME;
END_VAR
VAR
	tempArray :ARRAY [0..NUMBER_OF_SETS] OF TIME;
	temp :TIME;
	i :INT;
END_VAR
tempArray := inputArray;

FOR i := 0 TO (NUMBER_OF_SETS/2 - 1) DO
	temp := inputArray[i];
	tempArray[i] := inputArray[NUMBER_OF_SETS - i];
	tempArray[NUMBER_OF_SETS - i] := temp;
END_FOR

mirrorSimpleTimeArray := tempArray;
END_METHOD

(*

short summary
=============

.. <legal notes>

legal notes
=================
| SPDX-FileCopyrightText: © 2023 ekvip automation GmbH <info@ekvip.de>
| SPDX-License-Identifier: Apache-2.0
| For details check: Apache-2.0_

.. _Apache-2.0: https://www.apache.org/licenses/LICENSE-2.0

.. </legal notes>

parameters
==========

*)

{warning 'header is generated please add your documentation'}

METHOD testLongTimeHasExpired
VAR_INPUT
	currentValue :ARRAY [0..NUMBER_OF_SETS] OF LTIME;
	expectedValue :ARRAY [0..NUMBER_OF_SETS] OF LTIME;
END_VAR
VAR
	i :INT;
	message :Tc2_System.T_MaxString;
	timeStamp :LTIME;
	currentTime :LTIME;
	timeout :LTIME;
	timeExpired :BOOL;
END_VAR
VAR CONSTANT
	MAX_TIME :LTIME := TO_LTIME(16#FF_FF_FF_FF_FF_FF_FF_FF);
END_VAR

TEST('TEST--TimeAssertion--testLongTimeHasExpired');

FOR i := 0 TO 9 BY 1 DO
	
	THIS^.assertorContainer.resetAssertor();
	currentTime := LTIME();	
	timeStamp := SEL(currentTime > currentValue[i], currentTime - currentValue[i], currentTime);

	timeExpired := (TO_LINT(timeStamp)) >= (TO_LINT(currentTime));
	THIS^.assertorContainer.assertor.assert.times.long.timeHasExpired(
		timestamp := timeStamp,
		expiringTime := expectedValue[i],
		message := ''
	);
	
	
	
	message := 'TimeAssertionTests';
	message := Tc2_Standard.CONCAT(message, ' -> ');
	message := Tc2_Standard.CONCAT(message, 'longTimeHasExpired');
	message := Tc2_Standard.CONCAT(message, ' -> ');
	message := Tc2_Standard.CONCAT(message, ' Test ');
	message := Tc2_Standard.CONCAT(message, TO_STRING(i));
	message := Tc2_Standard.CONCAT(message, ' -> ');
	message := Tc2_Standard.CONCAT(message, ' currentValue = ');
	message := Tc2_Standard.CONCAT(message, TO_STRING(TO_LINT(currentValue[i])));	
	message := Tc2_Standard.CONCAT(message, ' -> ');
	message := Tc2_Standard.CONCAT(message, ' expectedValue = ');
	message := Tc2_Standard.CONCAT(message, TO_STRING(TO_LINT(expectedValue[i])));
	message := Tc2_Standard.CONCAT(message, ' -> ');
	message := Tc2_Standard.CONCAT(message, ' timestamp = ');
	message := Tc2_Standard.CONCAT(message, TO_STRING(TO_LINT(timeStamp)));
	message := Tc2_Standard.CONCAT(message, ' -> ');
	message := Tc2_Standard.CONCAT(message, ' currentTime = ');
	message := Tc2_Standard.CONCAT(message, TO_STRING(TO_LINT(currentTime)));
	message := Tc2_Standard.CONCAT(message, ' -> ');
	message := Tc2_Standard.CONCAT(message, ' timeExpired = ');
	message := Tc2_Standard.CONCAT(message, TO_STRING(TO_LINT(timeExpired)));
	message := Tc2_Standard.CONCAT(message, ' => ');
	message := Tc2_Standard.CONCAT(message, ' assertionWasWrong = ');
	message := Tc2_Standard.CONCAT(message, TO_STRING(THIS^.assertorContainer.wasAssertionWrong));



	IF (timeExpired) THEN
		THIS^.AssertFALSE(
			Condition := THIS^.assertorContainer.wasAssertionWrong,
			Message := message
		);
	ELSE
		THIS^.AssertTrue(
			Condition := THIS^.assertorContainer.wasAssertionWrong,
			Message := message
		);		
	END_IF
	
END_FOR;


TEST_FINISHED();
END_METHOD

(*

short summary
=============

.. <legal notes>

legal notes
=================
| SPDX-FileCopyrightText: © 2023 ekvip automation GmbH <info@ekvip.de>
| SPDX-License-Identifier: Apache-2.0
| For details check: Apache-2.0_

.. _Apache-2.0: https://www.apache.org/licenses/LICENSE-2.0

.. </legal notes>

parameters
==========

*)

{warning 'header is generated please add your documentation'}

METHOD testLongTimeHasNotExpired
VAR_INPUT
	currentValue :ARRAY [0..NUMBER_OF_SETS] OF LTIME;
	expectedValue :ARRAY [0..NUMBER_OF_SETS] OF LTIME;
END_VAR
VAR
	i :INT;
	message :Tc2_System.T_MaxString;
	 timeStamp :LTIME;
	 currentTime :LTIME;
	 timeout :LTIME;
	 timeExpired :BOOL;
END_VAR
VAR CONSTANT
	MAX_TIME :LTIME := TO_LTIME(16#FF_FF_FF_FF_FF_FF_FF_FF);
END_VAR

TEST('TEST--TimeAssertion--testLongTimeHasNotExpired');

FOR i := 0 TO 9 BY 1 DO
	
	THIS^.assertorContainer.resetAssertor();
	currentTime := LTIME();	
//	timeStamp := SEL(currentTime < currentValue[i], currentTime - currentValue[i], MAX_TIME - currentValue[i] + currentTime);
	timeStamp := SEL(currentTime > currentValue[i], currentTime - currentValue[i], currentTime);

	timeExpired := (TO_LINT(timeStamp)) >= (TO_LINT(currentTime));
	THIS^.assertorContainer.assertor.assert.times.long.timeHasNotExpired(
		timestamp := timeStamp,
		expiringTime := expectedValue[i],
		message := ''
	);
	
	
	
	message := 'TimeAssertionTests';
	message := Tc2_Standard.CONCAT(message, ' -> ');
	message := Tc2_Standard.CONCAT(message, 'longTimeHasNotExpired');
	message := Tc2_Standard.CONCAT(message, ' -> ');
	message := Tc2_Standard.CONCAT(message, ' Test ');
	message := Tc2_Standard.CONCAT(message, TO_STRING(i));
	message := Tc2_Standard.CONCAT(message, ' -> ');
	message := Tc2_Standard.CONCAT(message, ' currentValue = ');
	message := Tc2_Standard.CONCAT(message, TO_STRING(TO_LINT(currentValue[i])));	
	message := Tc2_Standard.CONCAT(message, ' -> ');
	message := Tc2_Standard.CONCAT(message, ' expectedValue = ');
	message := Tc2_Standard.CONCAT(message, TO_STRING(TO_LINT(expectedValue[i])));
	message := Tc2_Standard.CONCAT(message, ' -> ');
	message := Tc2_Standard.CONCAT(message, ' timestamp = ');
	message := Tc2_Standard.CONCAT(message, TO_STRING(TO_LINT(timeStamp)));
	message := Tc2_Standard.CONCAT(message, ' -> ');
	message := Tc2_Standard.CONCAT(message, ' currentTime = ');
	message := Tc2_Standard.CONCAT(message, TO_STRING(TO_LINT(currentTime)));
	message := Tc2_Standard.CONCAT(message, ' -> ');
	message := Tc2_Standard.CONCAT(message, ' timeExpired = ');
	message := Tc2_Standard.CONCAT(message, TO_STRING(TO_LINT(timeExpired)));
	message := Tc2_Standard.CONCAT(message, ' => ');
	message := Tc2_Standard.CONCAT(message, ' assertionWasWrong = ');
	message := Tc2_Standard.CONCAT(message, TO_STRING(THIS^.assertorContainer.wasAssertionWrong));


	IF (NOT timeExpired) THEN
		THIS^.AssertFALSE(
			Condition := THIS^.assertorContainer.wasAssertionWrong,
			Message := message
		);
	ELSE
		THIS^.AssertTrue(
			Condition := THIS^.assertorContainer.wasAssertionWrong,
			Message := message
		);		
	END_IF
	
END_FOR;


TEST_FINISHED();
END_METHOD

(*

short summary
=============

.. <legal notes>

legal notes
=================
| SPDX-FileCopyrightText: © 2023 ekvip automation GmbH <info@ekvip.de>
| SPDX-License-Identifier: Apache-2.0
| For details check: Apache-2.0_

.. _Apache-2.0: https://www.apache.org/licenses/LICENSE-2.0

.. </legal notes>

parameters
==========

*)

{warning 'header is generated please add your documentation'}

METHOD testLongValueIsEqualTo
VAR_INPUT
	currentValue :ARRAY [0..NUMBER_OF_SETS] OF LTIME;
	expectedValue :ARRAY [0..NUMBER_OF_SETS] OF LTIME;
END_VAR
VAR
	i :INT;
	message :Tc2_System.T_MaxString;
END_VAR
TEST('TEST--TimeAssertion--testLongValueIsEqualTo');

FOR i := 0 TO 9 BY 1 DO
	
	THIS^.assertorContainer.resetAssertor();
	THIS^.assertorContainer.assertor.assert.times.long.valueIsEqualTo(
		currentValue := currentValue[i],
		expectedValue := expectedValue[i],
		message := ''
	);
	
	
	message := 'TimeAssertionTests';
	message := Tc2_Standard.CONCAT(message, ' => ');
	message := Tc2_Standard.CONCAT(message, 'longTimeValuesIsEqualTo');
	message := Tc2_Standard.CONCAT(message, ' => ');
	message := Tc2_Standard.CONCAT(message, ' Test ');
	message := Tc2_Standard.CONCAT(message, TO_STRING(i));
	message := Tc2_Standard.CONCAT(message, ' => ');
	message := Tc2_Standard.CONCAT(message, ' assertion shall be wrong ');
	message := Tc2_Standard.CONCAT(message, ' => ');
	message := Tc2_Standard.CONCAT(message, ' currentValue = ');
	message := Tc2_Standard.CONCAT(message, TO_STRING(currentValue[i]));
	message := Tc2_Standard.CONCAT(message, ' expectedValue = ');
	message := Tc2_Standard.CONCAT(message, TO_STRING(expectedValue[i]));
	message := Tc2_Standard.CONCAT(message, ' => ');
	message := Tc2_Standard.CONCAT(message, ' assertionWasWrong = ');
	message := Tc2_Standard.CONCAT(message, TO_STRING(THIS^.assertorContainer.wasAssertionWrong));

	IF (currentValue[i] = expectedValue[i]) THEN
		THIS^.AssertFalse(
			Condition := THIS^.assertorContainer.wasAssertionWrong,
			Message := message
		);
	ELSE
		THIS^.AssertTrue(
			Condition := THIS^.assertorContainer.wasAssertionWrong,
			Message := message
		);		
	END_IF
	
END_FOR;


TEST_FINISHED();
END_METHOD

(*

short summary
=============

.. <legal notes>

legal notes
=================
| SPDX-FileCopyrightText: © 2023 ekvip automation GmbH <info@ekvip.de>
| SPDX-License-Identifier: Apache-2.0
| For details check: Apache-2.0_

.. _Apache-2.0: https://www.apache.org/licenses/LICENSE-2.0

.. </legal notes>

parameters
==========

*)

{warning 'header is generated please add your documentation'}

METHOD testLongValueIsGreaterThan
VAR_INPUT
	currentValue :ARRAY [0..NUMBER_OF_SETS] OF LTIME;
	expectedValue :ARRAY [0..NUMBER_OF_SETS] OF LTIME;
END_VAR
VAR
	i :INT;
	message :Tc2_System.T_MaxString;
END_VAR

TEST('TEST--TimeAssertion--testLongValueIsGreaterThan');

FOR i := 0 TO 9 BY 1 DO
	
	THIS^.assertorContainer.resetAssertor();
	THIS^.assertorContainer.assertor.assert.times.long.valueIsGreaterThan(
		currentValue := currentValue[i],
		lessValue := expectedValue[i],
		message := ''
	);
	
	
	message := 'TimeAssertionTests';
	message := Tc2_Standard.CONCAT(message, ' => ');
	message := Tc2_Standard.CONCAT(message, 'longTimeValueIsGreaterThan');
	message := Tc2_Standard.CONCAT(message, ' => ');
	message := Tc2_Standard.CONCAT(message, ' Test ');
	message := Tc2_Standard.CONCAT(message, TO_STRING(i));
	message := Tc2_Standard.CONCAT(message, ' => ');
	message := Tc2_Standard.CONCAT(message, ' assertion shall be wrong ');
	message := Tc2_Standard.CONCAT(message, ' => ');
	message := Tc2_Standard.CONCAT(message, ' currentValue = ');
	message := Tc2_Standard.CONCAT(message, TO_STRING(currentValue[i]));
	message := Tc2_Standard.CONCAT(message, ' expectedValue = ');
	message := Tc2_Standard.CONCAT(message, TO_STRING(expectedValue[i]));
	message := Tc2_Standard.CONCAT(message, ' => ');
	message := Tc2_Standard.CONCAT(message, ' assertionWasWrong = ');
	message := Tc2_Standard.CONCAT(message, TO_STRING(THIS^.assertorContainer.wasAssertionWrong));

	IF (currentValue[i] <= expectedValue[i]) THEN
		THIS^.AssertTrue(
			Condition := THIS^.assertorContainer.wasAssertionWrong,
			Message := message
		);
	ELSE
		THIS^.AssertFalse(
			Condition := THIS^.assertorContainer.wasAssertionWrong,
			Message := message
		);		
	END_IF
	
END_FOR;


TEST_FINISHED();
END_METHOD

(*

short summary
=============

.. <legal notes>

legal notes
=================
| SPDX-FileCopyrightText: © 2023 ekvip automation GmbH <info@ekvip.de>
| SPDX-License-Identifier: Apache-2.0
| For details check: Apache-2.0_

.. _Apache-2.0: https://www.apache.org/licenses/LICENSE-2.0

.. </legal notes>

parameters
==========

*)

{warning 'header is generated please add your documentation'}

METHOD testLongValueIsInRangeOf
VAR_INPUT
	currentValue :ARRAY [0..NUMBER_OF_SETS] OF LTIME;
	lowerLimit :ARRAY [0..NUMBER_OF_SETS] OF LTIME;
	upperLimit :ARRAY [0..NUMBER_OF_SETS] OF LTIME;
END_VAR
VAR
	i :INT;
	message :Tc2_System.T_MaxString;
END_VAR

TEST('TEST--TimeAssertion--testLongValueIsInRangeOf');

FOR i := 0 TO 9 BY 1 DO
	
	THIS^.assertorContainer.resetAssertor();
	THIS^.assertorContainer.assertor.assert.times.long.valueIsInRangeOf(
		currentValue := currentValue[i],
		lowerLimit := lowerLimit[i],
		upperLimit := upperLimit[i],
		message := ''
	);
	
	
	message := 'TimeAssertionTests';
	message := Tc2_Standard.CONCAT(message, ' => ');
	message := Tc2_Standard.CONCAT(message, 'testLongValueIsInRangeOf');
	message := Tc2_Standard.CONCAT(message, ' => ');
	message := Tc2_Standard.CONCAT(message, ' Test ');
	message := Tc2_Standard.CONCAT(message, TO_STRING(i));
	message := Tc2_Standard.CONCAT(message, ' => ');
	message := Tc2_Standard.CONCAT(message, ' assertion shall be wrong ');
	message := Tc2_Standard.CONCAT(message, ' => ');
	message := Tc2_Standard.CONCAT(message, ' currentValue = ');
	message := Tc2_Standard.CONCAT(message, TO_STRING(currentValue[i]));
	message := Tc2_Standard.CONCAT(message, ' => ');
	message := Tc2_Standard.CONCAT(message, ' lowerLimit = ');
	message := Tc2_Standard.CONCAT(message, TO_STRING(lowerLimit[i]));
	message := Tc2_Standard.CONCAT(message, ' => ');
	message := Tc2_Standard.CONCAT(message, ' upperLimit = ');
	message := Tc2_Standard.CONCAT(message, TO_STRING(upperLimit[i]));
	message := Tc2_Standard.CONCAT(message, ' => ');
	message := Tc2_Standard.CONCAT(message, ' assertionWasWrong = ');
	message := Tc2_Standard.CONCAT(message, TO_STRING(THIS^.assertorContainer.wasAssertionWrong));


	IF ((currentValue[i] >= lowerLimit[i]) AND (currentValue[i] <= upperLimit[i])) THEN
		THIS^.AssertFalse(
			Condition := THIS^.assertorContainer.wasAssertionWrong,
			Message := message
		);
	ELSE
		THIS^.AssertTrue(
			Condition := THIS^.assertorContainer.wasAssertionWrong,
			Message := message
		);		
	END_IF
	
END_FOR;


TEST_FINISHED();
END_METHOD

(*

short summary
=============

.. <legal notes>

legal notes
=================
| SPDX-FileCopyrightText: © 2023 ekvip automation GmbH <info@ekvip.de>
| SPDX-License-Identifier: Apache-2.0
| For details check: Apache-2.0_

.. _Apache-2.0: https://www.apache.org/licenses/LICENSE-2.0

.. </legal notes>

parameters
==========

*)

{warning 'header is generated please add your documentation'}

METHOD testLongValueIsLessThan
VAR_INPUT
	currentValue :ARRAY [0..NUMBER_OF_SETS] OF LTIME;
	expectedValue :ARRAY [0..NUMBER_OF_SETS] OF LTIME;
END_VAR
VAR
	i :INT;
	message :Tc2_System.T_MaxString;
END_VAR

TEST('TEST--TimeAssertion--testLongValueIsLessThan');

FOR i := 0 TO 9 BY 1 DO
	
	THIS^.assertorContainer.resetAssertor();
	THIS^.assertorContainer.assertor.assert.times.long.valueIsLessThan(
		currentValue := currentValue[i],
		greaterValue := expectedValue[i],
		message := ''
	);
	
	
	message := 'TimeAssertionTests';
	message := Tc2_Standard.CONCAT(message, ' => ');
	message := Tc2_Standard.CONCAT(message, ' longTimeValueIslessThan');
	message := Tc2_Standard.CONCAT(message, ' => ');
	message := Tc2_Standard.CONCAT(message, ' Test ');
	message := Tc2_Standard.CONCAT(message, TO_STRING(i));
	message := Tc2_Standard.CONCAT(message, ' => ');
	message := Tc2_Standard.CONCAT(message, ' assertion shall be wrong ');
	message := Tc2_Standard.CONCAT(message, ' => ');
	message := Tc2_Standard.CONCAT(message, ' currentValue = ');
	message := Tc2_Standard.CONCAT(message, TO_STRING(currentValue[i]));
	message := Tc2_Standard.CONCAT(message, ' expectedValue = ');
	message := Tc2_Standard.CONCAT(message, TO_STRING(expectedValue[i]));
	message := Tc2_Standard.CONCAT(message, ' => ');
	message := Tc2_Standard.CONCAT(message, ' assertionWasWrong = ');
	message := Tc2_Standard.CONCAT(message, TO_STRING(THIS^.assertorContainer.wasAssertionWrong));


	IF (currentValue[i] >= expectedValue[i]) THEN
		THIS^.AssertTrue(
			Condition := THIS^.assertorContainer.wasAssertionWrong,
			Message := message
		);
	ELSE
		THIS^.AssertFalse(
			Condition := THIS^.assertorContainer.wasAssertionWrong,
			Message := message
		);		
	END_IF
	
END_FOR;


TEST_FINISHED();
END_METHOD

(*

short summary
=============

.. <legal notes>

legal notes
=================
| SPDX-FileCopyrightText: © 2023 ekvip automation GmbH <info@ekvip.de>
| SPDX-License-Identifier: Apache-2.0
| For details check: Apache-2.0_

.. _Apache-2.0: https://www.apache.org/licenses/LICENSE-2.0

.. </legal notes>

parameters
==========

*)

{warning 'header is generated please add your documentation'}

METHOD testLongValueIsMax
VAR_INPUT
	currentValue :ARRAY [0..NUMBER_OF_SETS] OF LTIME;
	expectedValue :ARRAY [0..NUMBER_OF_SETS] OF LTIME;
END_VAR
VAR
	i :INT;
	message :Tc2_System.T_MaxString;
END_VAR

TEST('TEST--TimeAssertion--testLongValueIsMax');

FOR i := 0 TO 9 BY 1 DO
	
	THIS^.assertorContainer.resetAssertor();
	THIS^.assertorContainer.assertor.assert.times.long.valueIsMax(
		currentValue := currentValue[i],
		maximumValue := expectedValue[i],
		message := ''
	);
	
	
	message := 'TimeAssertionTests';
	message := Tc2_Standard.CONCAT(message, ' => ');
	message := Tc2_Standard.CONCAT(message, 'longTimeValueIsMax');
	message := Tc2_Standard.CONCAT(message, ' => ');
	message := Tc2_Standard.CONCAT(message, ' Test ');
	message := Tc2_Standard.CONCAT(message, TO_STRING(i));
	message := Tc2_Standard.CONCAT(message, ' => ');
	message := Tc2_Standard.CONCAT(message, ' assertion shall be wrong ');
	message := Tc2_Standard.CONCAT(message, ' => ');
	message := Tc2_Standard.CONCAT(message, ' currentValue = ');
	message := Tc2_Standard.CONCAT(message, TO_STRING(currentValue[i]));
	message := Tc2_Standard.CONCAT(message, ' expectedValue = ');
	message := Tc2_Standard.CONCAT(message, TO_STRING(expectedValue[i]));

	IF (currentValue[i] <= expectedValue[i]) THEN
		THIS^.AssertFalse(
			Condition := THIS^.assertorContainer.wasAssertionWrong,
			Message := message
		);
	ELSE
		THIS^.AssertTrue(
			Condition := THIS^.assertorContainer.wasAssertionWrong,
			Message := message
		);		
	END_IF
	
END_FOR;


TEST_FINISHED();
END_METHOD

(*

short summary
=============

.. <legal notes>

legal notes
=================
| SPDX-FileCopyrightText: © 2023 ekvip automation GmbH <info@ekvip.de>
| SPDX-License-Identifier: Apache-2.0
| For details check: Apache-2.0_

.. _Apache-2.0: https://www.apache.org/licenses/LICENSE-2.0

.. </legal notes>

parameters
==========

*)

{warning 'header is generated please add your documentation'}

METHOD testLongValueIsMin
VAR_INPUT
	currentValue :ARRAY [0..NUMBER_OF_SETS] OF LTIME;
	expectedValue :ARRAY [0..NUMBER_OF_SETS] OF LTIME;
END_VAR
VAR
	i :INT;
	message :Tc2_System.T_MaxString;
END_VAR

TEST('TEST--TimeAssertion--testLongValueIsMin');

FOR i := 0 TO 9 BY 1 DO
	
	THIS^.assertorContainer.resetAssertor();
	THIS^.assertorContainer.assertor.assert.times.long.valueIsMin(
		currentValue := currentValue[i],
		minimumValue := expectedValue[i],
		message := ''
	);
	
	
	message := 'TimeAssertionTests';
	message := Tc2_Standard.CONCAT(message, ' => ');
	message := Tc2_Standard.CONCAT(message, 'longTimeValueIsMin');
	message := Tc2_Standard.CONCAT(message, ' => ');
	message := Tc2_Standard.CONCAT(message, ' Test ');
	message := Tc2_Standard.CONCAT(message, TO_STRING(i));
	message := Tc2_Standard.CONCAT(message, ' => ');
	message := Tc2_Standard.CONCAT(message, ' assertion shall be wrong ');
	message := Tc2_Standard.CONCAT(message, ' => ');
	message := Tc2_Standard.CONCAT(message, ' currentValue = ');
	message := Tc2_Standard.CONCAT(message, TO_STRING(currentValue[i]));
	message := Tc2_Standard.CONCAT(message, ' expectedValue = ');
	message := Tc2_Standard.CONCAT(message, TO_STRING(expectedValue[i]));

	IF (currentValue[i] >= expectedValue[i]) THEN
		THIS^.AssertFalse(
			Condition := THIS^.assertorContainer.wasAssertionWrong,
			Message := message
		);
	ELSE
		THIS^.AssertTrue(
			Condition := THIS^.assertorContainer.wasAssertionWrong,
			Message := message
		);		
	END_IF
	
END_FOR;


TEST_FINISHED();
END_METHOD

(*

short summary
=============

.. <legal notes>

legal notes
=================
| SPDX-FileCopyrightText: © 2023 ekvip automation GmbH <info@ekvip.de>
| SPDX-License-Identifier: Apache-2.0
| For details check: Apache-2.0_

.. _Apache-2.0: https://www.apache.org/licenses/LICENSE-2.0

.. </legal notes>

parameters
==========

*)

{warning 'header is generated please add your documentation'}

METHOD testLongValueIsNotEqualTo
VAR_INPUT
	currentValue :ARRAY [0..NUMBER_OF_SETS] OF LTIME;
	expectedValue :ARRAY [0..NUMBER_OF_SETS] OF LTIME;
END_VAR
VAR
	i :INT;
	message :Tc2_System.T_MaxString;
END_VAR

TEST('TEST--TimeAssertion--testLongValueIsNotEqualTo');

FOR i := 0 TO 9 BY 1 DO
	
	THIS^.assertorContainer.resetAssertor();
	THIS^.assertorContainer.assertor.assert.times.long.valueIsNotEqualTo(
		currentValue := currentValue[i],
		unexpectedValue := expectedValue[i],
		message := ''
	);
	
	message := 'TimeAssertionTests';
	message := Tc2_Standard.CONCAT(message, ' => ');
	message := Tc2_Standard.CONCAT(message, ' longTimeValuesIsNotEqualTo');
	message := Tc2_Standard.CONCAT(message, ' Test ');
	message := Tc2_Standard.CONCAT(message, TO_STRING(i));
	message := Tc2_Standard.CONCAT(message, ' => ');
	message := Tc2_Standard.CONCAT(message, ' assertion shall be wrong ');
	message := Tc2_Standard.CONCAT(message, ' => ');
	message := Tc2_Standard.CONCAT(message, ' currentValue = ');
	message := Tc2_Standard.CONCAT(message, TO_STRING(currentValue[i]));
	message := Tc2_Standard.CONCAT(message, ' expectedValue = ');
	message := Tc2_Standard.CONCAT(message, TO_STRING(expectedValue[i]));

	IF (currentValue[i] <> expectedValue[i]) THEN
		THIS^.AssertFalse(
			Condition := THIS^.assertorContainer.wasAssertionWrong,
			Message := message
		);
	ELSE
		THIS^.AssertTrue(
			Condition := THIS^.assertorContainer.wasAssertionWrong,
			Message := message
		);		
	END_IF
	
END_FOR;


TEST_FINISHED();
END_METHOD

(*

short summary
=============

.. <legal notes>

legal notes
=================
| SPDX-FileCopyrightText: © 2023 ekvip automation GmbH <info@ekvip.de>
| SPDX-License-Identifier: Apache-2.0
| For details check: Apache-2.0_

.. _Apache-2.0: https://www.apache.org/licenses/LICENSE-2.0

.. </legal notes>

parameters
==========

*)

{warning 'header is generated please add your documentation'}

METHOD testSimpleTimeHasExpired
VAR_INPUT
	currentValue :ARRAY [0..NUMBER_OF_SETS] OF TIME;
	expectedValue :ARRAY [0..NUMBER_OF_SETS] OF TIME;
END_VAR
VAR
	i :INT;
	message :Tc2_System.T_MaxString;
	 timeStamp :TIME;
	 currentTime :TIME;
	 timeout :TIME;
	 timeExpired :BOOL;
END_VAR
VAR CONSTANT
	MAX_TIME :TIME := TO_TIME(16#FF_FF_FF_FF);
END_VAR

TEST('TEST--TimeAssertion--time has expired');

FOR i := 0 TO 9 BY 1 DO
	
	THIS^.assertorContainer.resetAssertor();
	currentTime := TIME();	
//	timeStamp := SEL(currentTime < currentValue[i], currentTime - currentValue[i], MAX_TIME - currentValue[i] + currentTime);
	timeStamp := SEL(currentTime > currentValue[i], currentTime - currentValue[i], currentTime);

	timeExpired := (TO_LINT(timeStamp)) >= (TO_LINT(currentTime));
	THIS^.assertorContainer.assertor.assert.times.simple.timeHasExpired(
		timestamp := timeStamp,
		expiringTime := expectedValue[i],
		message := ''
	);
	
	
	
	message := 'TimeAssertionTests';
	message := Tc2_Standard.CONCAT(message, ' -> ');
	message := Tc2_Standard.CONCAT(message, 'simpleTimeHasExpired');
	message := Tc2_Standard.CONCAT(message, ' -> ');
	message := Tc2_Standard.CONCAT(message, ' Test ');
	message := Tc2_Standard.CONCAT(message, TO_STRING(i));
	message := Tc2_Standard.CONCAT(message, ' -> ');
	message := Tc2_Standard.CONCAT(message, ' currentValue = ');
	message := Tc2_Standard.CONCAT(message, TO_STRING(TO_LINT(currentValue[i])));	
	message := Tc2_Standard.CONCAT(message, ' -> ');
	message := Tc2_Standard.CONCAT(message, ' expectedValue = ');
	message := Tc2_Standard.CONCAT(message, TO_STRING(TO_LINT(expectedValue[i])));
	message := Tc2_Standard.CONCAT(message, ' -> ');
	message := Tc2_Standard.CONCAT(message, ' timestamp = ');
	message := Tc2_Standard.CONCAT(message, TO_STRING(TO_LINT(timeStamp)));
	message := Tc2_Standard.CONCAT(message, ' -> ');
	message := Tc2_Standard.CONCAT(message, ' currentTime = ');
	message := Tc2_Standard.CONCAT(message, TO_STRING(TO_LINT(currentTime)));
	message := Tc2_Standard.CONCAT(message, ' -> ');
	message := Tc2_Standard.CONCAT(message, ' timeExpired = ');
	message := Tc2_Standard.CONCAT(message, TO_STRING(TO_LINT(timeExpired)));


	IF (timeExpired) THEN
		THIS^.AssertFALSE(
			Condition := THIS^.assertorContainer.wasAssertionWrong,
			Message := message
		);
	ELSE
		THIS^.AssertTrue(
			Condition := THIS^.assertorContainer.wasAssertionWrong,
			Message := message
		);		
	END_IF
	
END_FOR;


TEST_FINISHED();
END_METHOD

(*

short summary
=============

.. <legal notes>

legal notes
=================
| SPDX-FileCopyrightText: © 2023 ekvip automation GmbH <info@ekvip.de>
| SPDX-License-Identifier: Apache-2.0
| For details check: Apache-2.0_

.. _Apache-2.0: https://www.apache.org/licenses/LICENSE-2.0

.. </legal notes>

parameters
==========

*)

{warning 'header is generated please add your documentation'}

METHOD testSimpleTimeHasNotExpired
VAR_INPUT
	currentValue :ARRAY [0..NUMBER_OF_SETS] OF TIME;
	expectedValue :ARRAY [0..NUMBER_OF_SETS] OF TIME;
END_VAR
VAR
	i :INT;
	message :Tc2_System.T_MaxString;
	 timeStamp :TIME;
	 currentTime :TIME;
	 timeout :TIME;
	 timeExpired :BOOL;
END_VAR
VAR CONSTANT
	MAX_TIME :TIME := TO_TIME(16#FF_FF_FF_FF);
END_VAR

TEST('TEST--TimeAssertion--testSimpleTimeHasNotExpired');

FOR i := 0 TO 9 BY 1 DO
	
	THIS^.assertorContainer.resetAssertor();
	currentTime := TIME();	
//	timeStamp := SEL(currentTime < currentValue[i], currentTime - currentValue[i], MAX_TIME - currentValue[i] + currentTime);
	timeStamp := SEL(currentTime > currentValue[i], currentTime - currentValue[i], currentTime);

	timeExpired := (TO_LINT(timeStamp)) >= (TO_LINT(currentTime));
	THIS^.assertorContainer.assertor.assert.times.simple.timeHasNotExpired(
		timestamp := timeStamp,
		expiringTime := expectedValue[i],
		message := ''
	);
	
	
	
	message := 'TimeAssertionTests';
	message := Tc2_Standard.CONCAT(message, ' -> ');
	message := Tc2_Standard.CONCAT(message, 'simpleTimeHasNotExpired');
	message := Tc2_Standard.CONCAT(message, ' -> ');
	message := Tc2_Standard.CONCAT(message, ' Test ');
	message := Tc2_Standard.CONCAT(message, TO_STRING(i));
	message := Tc2_Standard.CONCAT(message, ' -> ');
	message := Tc2_Standard.CONCAT(message, ' currentValue = ');
	message := Tc2_Standard.CONCAT(message, TO_STRING(TO_LINT(currentValue[i])));	
	message := Tc2_Standard.CONCAT(message, ' -> ');
	message := Tc2_Standard.CONCAT(message, ' expectedValue = ');
	message := Tc2_Standard.CONCAT(message, TO_STRING(TO_LINT(expectedValue[i])));
	message := Tc2_Standard.CONCAT(message, ' -> ');
	message := Tc2_Standard.CONCAT(message, ' timestamp = ');
	message := Tc2_Standard.CONCAT(message, TO_STRING(TO_LINT(timeStamp)));
	message := Tc2_Standard.CONCAT(message, ' -> ');
	message := Tc2_Standard.CONCAT(message, ' currentTime = ');
	message := Tc2_Standard.CONCAT(message, TO_STRING(TO_LINT(currentTime)));
	message := Tc2_Standard.CONCAT(message, ' -> ');
	message := Tc2_Standard.CONCAT(message, ' timeExpired = ');
	message := Tc2_Standard.CONCAT(message, TO_STRING(TO_LINT(timeExpired)));


	IF (NOT timeExpired) THEN
		THIS^.AssertFALSE(
			Condition := THIS^.assertorContainer.wasAssertionWrong,
			Message := message
		);
	ELSE
		THIS^.AssertTrue(
			Condition := THIS^.assertorContainer.wasAssertionWrong,
			Message := message
		);		
	END_IF
	
END_FOR;


TEST_FINISHED();
END_METHOD

(*

short summary
=============

.. <legal notes>

legal notes
=================
| SPDX-FileCopyrightText: © 2023 ekvip automation GmbH <info@ekvip.de>
| SPDX-License-Identifier: Apache-2.0
| For details check: Apache-2.0_

.. _Apache-2.0: https://www.apache.org/licenses/LICENSE-2.0

.. </legal notes>

parameters
==========

*)

{warning 'header is generated please add your documentation'}

METHOD testSimpleValueIsEqualTo
VAR_INPUT
	currentValue :ARRAY [0..NUMBER_OF_SETS] OF TIME;
	expectedValue :ARRAY [0..NUMBER_OF_SETS] OF TIME;
END_VAR
VAR
	i :INT;
	message :Tc2_System.T_MaxString;
END_VAR
TEST('TEST--TimeAssertion--testSimpleValueIsEqualTo');

FOR i := 0 TO 9 BY 1 DO
	
	THIS^.assertorContainer.resetAssertor();
	THIS^.assertorContainer.assertor.assert.times.simple.valueIsEqualTo(
		currentValue := currentValue[i],
		expectedValue := expectedValue[i],
		message := ''
	);
	
	
	message := 'TimeAssertionTests';
	message := Tc2_Standard.CONCAT(message, ' => ');
	message := Tc2_Standard.CONCAT(message, 'simpleTimeValuesIsEqualTo');
	message := Tc2_Standard.CONCAT(message, ' => ');
	message := Tc2_Standard.CONCAT(message, ' Test ');
	message := Tc2_Standard.CONCAT(message, TO_STRING(i));
	message := Tc2_Standard.CONCAT(message, ' => ');
	message := Tc2_Standard.CONCAT(message, ' assertion shall be wrong ');
	message := Tc2_Standard.CONCAT(message, ' => ');
	message := Tc2_Standard.CONCAT(message, ' currentValue = ');
	message := Tc2_Standard.CONCAT(message, TO_STRING(currentValue[i]));
	message := Tc2_Standard.CONCAT(message, ' expectedValue = ');
	message := Tc2_Standard.CONCAT(message, TO_STRING(expectedValue[i]));

	IF (currentValue[i] = expectedValue[i]) THEN
		THIS^.AssertFalse(
			Condition := THIS^.assertorContainer.wasAssertionWrong,
			Message := message
		);
	ELSE
		THIS^.AssertTrue(
			Condition := THIS^.assertorContainer.wasAssertionWrong,
			Message := message
		);		
	END_IF
	
END_FOR;


TEST_FINISHED();
END_METHOD

(*

short summary
=============

.. <legal notes>

legal notes
=================
| SPDX-FileCopyrightText: © 2023 ekvip automation GmbH <info@ekvip.de>
| SPDX-License-Identifier: Apache-2.0
| For details check: Apache-2.0_

.. _Apache-2.0: https://www.apache.org/licenses/LICENSE-2.0

.. </legal notes>

parameters
==========

*)

{warning 'header is generated please add your documentation'}

METHOD testSimpleValueIsGreaterThan
VAR_INPUT
	currentValue :ARRAY [0..NUMBER_OF_SETS] OF TIME;
	expectedValue :ARRAY [0..NUMBER_OF_SETS] OF TIME;
END_VAR
VAR
	i :INT;
	message :Tc2_System.T_MaxString;
END_VAR
TEST('TEST--TimeAssertion--testSimpleValueIsGreaterThan');

FOR i := 0 TO 9 BY 1 DO
	
	THIS^.assertorContainer.resetAssertor();
	THIS^.assertorContainer.assertor.assert.times.simple.valueIsGreaterThan(
		currentValue := currentValue[i],
		lessValue := expectedValue[i],
		message := ''
	);
	
	
	message := 'TimeAssertionTests';
	message := Tc2_Standard.CONCAT(message, ' => ');
	message := Tc2_Standard.CONCAT(message, 'simpleTimeValueIsGreaterThan');
	message := Tc2_Standard.CONCAT(message, ' => ');
	message := Tc2_Standard.CONCAT(message, ' Test ');
	message := Tc2_Standard.CONCAT(message, TO_STRING(i));
	message := Tc2_Standard.CONCAT(message, ' => ');
	message := Tc2_Standard.CONCAT(message, ' assertion shall be wrong ');
	message := Tc2_Standard.CONCAT(message, ' => ');
	message := Tc2_Standard.CONCAT(message, ' currentValue = ');
	message := Tc2_Standard.CONCAT(message, TO_STRING(currentValue[i]));
	message := Tc2_Standard.CONCAT(message, ' expectedValue = ');
	message := Tc2_Standard.CONCAT(message, TO_STRING(expectedValue[i]));

	IF (currentValue[i] <= expectedValue[i]) THEN
		THIS^.AssertTrue(
			Condition := THIS^.assertorContainer.wasAssertionWrong,
			Message := message
		);
	ELSE
		THIS^.AssertFalse(
			Condition := THIS^.assertorContainer.wasAssertionWrong,
			Message := message
		);		
	END_IF
	
END_FOR;


TEST_FINISHED();
END_METHOD

(*

short summary
=============

.. <legal notes>

legal notes
=================
| SPDX-FileCopyrightText: © 2023 ekvip automation GmbH <info@ekvip.de>
| SPDX-License-Identifier: Apache-2.0
| For details check: Apache-2.0_

.. _Apache-2.0: https://www.apache.org/licenses/LICENSE-2.0

.. </legal notes>

parameters
==========

*)

{warning 'header is generated please add your documentation'}

METHOD testSimpleValueIsInRangeOf
VAR_INPUT
	currentValue :ARRAY [0..NUMBER_OF_SETS] OF TIME;
	lowerLimit :ARRAY [0..NUMBER_OF_SETS] OF TIME;
	upperLimit :ARRAY [0..NUMBER_OF_SETS] OF TIME;
END_VAR
VAR
	i :INT;
	message :Tc2_System.T_MaxString;
END_VAR
TEST('TEST--TimeAssertion--testSimpleValueIsInRangeOf');

FOR i := 0 TO 9 BY 1 DO
	
	THIS^.assertorContainer.resetAssertor();
	THIS^.assertorContainer.assertor.assert.times.simple.valueIsInRangeOf(
		currentValue := currentValue[i],
		lowerLimit := lowerLimit[i],
		upperLimit := upperLimit[i],
		message := ''
	);
	
	
	message := 'TimeAssertionTests';
	message := Tc2_Standard.CONCAT(message, ' => ');
	message := Tc2_Standard.CONCAT(message, 'testSimpleValueIsInRangeOf');
	message := Tc2_Standard.CONCAT(message, ' => ');
	message := Tc2_Standard.CONCAT(message, ' Test ');
	message := Tc2_Standard.CONCAT(message, TO_STRING(i));
	message := Tc2_Standard.CONCAT(message, ' => ');
	message := Tc2_Standard.CONCAT(message, ' assertion shall be wrong ');
	message := Tc2_Standard.CONCAT(message, ' => ');
	message := Tc2_Standard.CONCAT(message, ' currentValue = ');
	message := Tc2_Standard.CONCAT(message, TO_STRING(currentValue[i]));
	message := Tc2_Standard.CONCAT(message, ' => ');
	message := Tc2_Standard.CONCAT(message, ' lowerLimit = ');
	message := Tc2_Standard.CONCAT(message, TO_STRING(lowerLimit[i]));
	message := Tc2_Standard.CONCAT(message, ' => ');
	message := Tc2_Standard.CONCAT(message, ' upperLimit = ');
	message := Tc2_Standard.CONCAT(message, TO_STRING(upperLimit[i]));
	message := Tc2_Standard.CONCAT(message, ' => ');
	message := Tc2_Standard.CONCAT(message, ' assertionWasWrong = ');
	message := Tc2_Standard.CONCAT(message, TO_STRING(THIS^.assertorContainer.wasAssertionWrong));


	IF ((currentValue[i] >= lowerLimit[i]) AND (currentValue[i] <= upperLimit[i])) THEN
		THIS^.AssertFalse(
			Condition := THIS^.assertorContainer.wasAssertionWrong,
			Message := message
		);
	ELSE
		THIS^.AssertTrue(
			Condition := THIS^.assertorContainer.wasAssertionWrong,
			Message := message
		);		
	END_IF
	
END_FOR;


TEST_FINISHED();
END_METHOD

(*

short summary
=============

.. <legal notes>

legal notes
=================
| SPDX-FileCopyrightText: © 2023 ekvip automation GmbH <info@ekvip.de>
| SPDX-License-Identifier: Apache-2.0
| For details check: Apache-2.0_

.. _Apache-2.0: https://www.apache.org/licenses/LICENSE-2.0

.. </legal notes>

parameters
==========

*)

{warning 'header is generated please add your documentation'}

METHOD testSimpleValueIsLessThan
VAR_INPUT
	currentValue :ARRAY [0..NUMBER_OF_SETS] OF TIME;
	expectedValue :ARRAY [0..NUMBER_OF_SETS] OF TIME;
END_VAR
VAR
	i :INT;
	message :Tc2_System.T_MaxString;
END_VAR
TEST('TEST--TimeAssertion--testSimpleValueIsLessThan');

FOR i := 0 TO 9 BY 1 DO
	
	THIS^.assertorContainer.resetAssertor();
	THIS^.assertorContainer.assertor.assert.times.simple.valueIsLessThan(
		currentValue := currentValue[i],
		greaterValue := expectedValue[i],
		message := ''
	);
	
	
	message := 'TimeAssertionTests';
	message := Tc2_Standard.CONCAT(message, ' => ');
	message := Tc2_Standard.CONCAT(message, 'simpleTimeValueIslessThan');
	message := Tc2_Standard.CONCAT(message, ' => ');
	message := Tc2_Standard.CONCAT(message, ' Test ');
	message := Tc2_Standard.CONCAT(message, TO_STRING(i));
	message := Tc2_Standard.CONCAT(message, ' => ');
	message := Tc2_Standard.CONCAT(message, ' assertion shall be wrong ');
	message := Tc2_Standard.CONCAT(message, ' => ');
	message := Tc2_Standard.CONCAT(message, ' currentValue = ');
	message := Tc2_Standard.CONCAT(message, TO_STRING(currentValue[i]));
	message := Tc2_Standard.CONCAT(message, ' expectedValue = ');
	message := Tc2_Standard.CONCAT(message, TO_STRING(expectedValue[i]));

	IF (currentValue[i] >= expectedValue[i]) THEN
		THIS^.AssertTrue(
			Condition := THIS^.assertorContainer.wasAssertionWrong,
			Message := message
		);
	ELSE
		THIS^.AssertFalse(
			Condition := THIS^.assertorContainer.wasAssertionWrong,
			Message := message
		);		
	END_IF
	
END_FOR;


TEST_FINISHED();
END_METHOD

(*

short summary
=============

.. <legal notes>

legal notes
=================
| SPDX-FileCopyrightText: © 2023 ekvip automation GmbH <info@ekvip.de>
| SPDX-License-Identifier: Apache-2.0
| For details check: Apache-2.0_

.. _Apache-2.0: https://www.apache.org/licenses/LICENSE-2.0

.. </legal notes>

parameters
==========

*)

{warning 'header is generated please add your documentation'}

METHOD testSimpleValueIsMax
VAR_INPUT
	currentValue :ARRAY [0..NUMBER_OF_SETS] OF TIME;
	expectedValue :ARRAY [0..NUMBER_OF_SETS] OF TIME;
END_VAR
VAR
	i :INT;
	message :Tc2_System.T_MaxString;
END_VAR
TEST('TEST--TimeAssertion--testSimpleValueIsMax');

FOR i := 0 TO 9 BY 1 DO
	
	THIS^.assertorContainer.resetAssertor();
	THIS^.assertorContainer.assertor.assert.times.simple.valueIsMax(
		currentValue := currentValue[i],
		maximumValue := expectedValue[i],
		message := ''
	);
	
	
	message := 'TimeAssertionTests';
	message := Tc2_Standard.CONCAT(message, ' => ');
	message := Tc2_Standard.CONCAT(message, 'simpleTimeValueIsMax');
	message := Tc2_Standard.CONCAT(message, ' => ');
	message := Tc2_Standard.CONCAT(message, ' Test ');
	message := Tc2_Standard.CONCAT(message, TO_STRING(i));
	message := Tc2_Standard.CONCAT(message, ' => ');
	message := Tc2_Standard.CONCAT(message, ' assertion shall be wrong ');
	message := Tc2_Standard.CONCAT(message, ' => ');
	message := Tc2_Standard.CONCAT(message, ' currentValue = ');
	message := Tc2_Standard.CONCAT(message, TO_STRING(currentValue[i]));
	message := Tc2_Standard.CONCAT(message, ' expectedValue = ');
	message := Tc2_Standard.CONCAT(message, TO_STRING(expectedValue[i]));

	IF (currentValue[i] <= expectedValue[i]) THEN
		THIS^.AssertFalse(
			Condition := THIS^.assertorContainer.wasAssertionWrong,
			Message := message
		);
	ELSE
		THIS^.AssertTrue(
			Condition := THIS^.assertorContainer.wasAssertionWrong,
			Message := message
		);		
	END_IF
	
END_FOR;


TEST_FINISHED();
END_METHOD

(*

short summary
=============

.. <legal notes>

legal notes
=================
| SPDX-FileCopyrightText: © 2023 ekvip automation GmbH <info@ekvip.de>
| SPDX-License-Identifier: Apache-2.0
| For details check: Apache-2.0_

.. _Apache-2.0: https://www.apache.org/licenses/LICENSE-2.0

.. </legal notes>

parameters
==========

*)

{warning 'header is generated please add your documentation'}

METHOD testSimpleValueIsMin
VAR_INPUT
	currentValue :ARRAY [0..NUMBER_OF_SETS] OF TIME;
	expectedValue :ARRAY [0..NUMBER_OF_SETS] OF TIME;
END_VAR
VAR
	i :INT;
	message :Tc2_System.T_MaxString;
END_VAR
TEST('TEST--TimeAssertion--testSimpleValueIsMin');

FOR i := 0 TO 9 BY 1 DO
	
	THIS^.assertorContainer.resetAssertor();
	THIS^.assertorContainer.assertor.assert.times.simple.valueIsMin(
		currentValue := currentValue[i],
		minimumValue := expectedValue[i],
		message := ''
	);
	
	
	message := 'TimeAssertionTests';
	message := Tc2_Standard.CONCAT(message, ' => ');
	message := Tc2_Standard.CONCAT(message, 'simpleTimeValueIsMin');
	message := Tc2_Standard.CONCAT(message, ' => ');
	message := Tc2_Standard.CONCAT(message, ' Test ');
	message := Tc2_Standard.CONCAT(message, TO_STRING(i));
	message := Tc2_Standard.CONCAT(message, ' => ');
	message := Tc2_Standard.CONCAT(message, ' assertion shall be wrong ');
	message := Tc2_Standard.CONCAT(message, ' => ');
	message := Tc2_Standard.CONCAT(message, ' currentValue = ');
	message := Tc2_Standard.CONCAT(message, TO_STRING(currentValue[i]));
	message := Tc2_Standard.CONCAT(message, ' expectedValue = ');
	message := Tc2_Standard.CONCAT(message, TO_STRING(expectedValue[i]));

	IF (currentValue[i] >= expectedValue[i]) THEN
		THIS^.AssertFalse(
			Condition := THIS^.assertorContainer.wasAssertionWrong,
			Message := message
		);
	ELSE
		THIS^.AssertTrue(
			Condition := THIS^.assertorContainer.wasAssertionWrong,
			Message := message
		);		
	END_IF
	
END_FOR;


TEST_FINISHED();
END_METHOD

(*

short summary
=============

.. <legal notes>

legal notes
=================
| SPDX-FileCopyrightText: © 2023 ekvip automation GmbH <info@ekvip.de>
| SPDX-License-Identifier: Apache-2.0
| For details check: Apache-2.0_

.. _Apache-2.0: https://www.apache.org/licenses/LICENSE-2.0

.. </legal notes>

parameters
==========

*)

{warning 'header is generated please add your documentation'}

METHOD testSimpleValueIsNotEqualTo
VAR_INPUT
	currentValue :ARRAY [0..NUMBER_OF_SETS] OF TIME;
	expectedValue :ARRAY [0..NUMBER_OF_SETS] OF TIME;
END_VAR
VAR
	i :INT;
	message :Tc2_System.T_MaxString;
END_VAR
TEST('TEST--TimeAssertion--testSimpleValueIsNotEqualTo');

FOR i := 0 TO 9 BY 1 DO
	
	THIS^.assertorContainer.resetAssertor();
	THIS^.assertorContainer.assertor.assert.times.simple.valueIsNotEqualTo(
		currentValue := currentValue[i],
		unexpectedValue := expectedValue[i],
		message := ''
	);
	
	message := 'TimeAssertionTests';
	message := Tc2_Standard.CONCAT(message, ' => ');
	message := Tc2_Standard.CONCAT(message, 'simpleTimeValuesIsNotEqualTo');
	message := Tc2_Standard.CONCAT(message, ' Test ');
	message := Tc2_Standard.CONCAT(message, TO_STRING(i));
	message := Tc2_Standard.CONCAT(message, ' => ');
	message := Tc2_Standard.CONCAT(message, ' assertion shall be wrong ');
	message := Tc2_Standard.CONCAT(message, ' => ');
	message := Tc2_Standard.CONCAT(message, ' currentValue = ');
	message := Tc2_Standard.CONCAT(message, TO_STRING(currentValue[i]));
	message := Tc2_Standard.CONCAT(message, ' expectedValue = ');
	message := Tc2_Standard.CONCAT(message, TO_STRING(expectedValue[i]));

	IF (currentValue[i] = expectedValue[i]) THEN
		THIS^.AssertTrue(
			Condition := THIS^.assertorContainer.wasAssertionWrong,
			Message := message
		);
	ELSE
		THIS^.AssertFalse(
			Condition := THIS^.assertorContainer.wasAssertionWrong,
			Message := message
		);		
	END_IF
	
END_FOR;


TEST_FINISHED();
END_METHOD

END_FUNCTION_BLOCK

// ---- AssertionTester/classes/AssertionTester.TcPOU
(*

short summary
=============

.. <legal notes>

legal notes
=================
| SPDX-FileCopyrightText: © 2023 ekvip automation GmbH <info@ekvip.de>
| SPDX-License-Identifier: Apache-2.0
| For details check: Apache-2.0_

.. _Apache-2.0: https://www.apache.org/licenses/LICENSE-2.0

.. </legal notes>

methods and properties
======================

*)

{warning 'header is generated please add your documentation'}
FUNCTION_BLOCK AssertionTester EXTENDS CNM_AbstractObject.Object IMPLEMENTS IAttachAssertorContainer
VAR	
	pointerTests 			:PointerAssertionsTests(classToBeTested := 0);
	uxintAssertions			:UxintAssertionTests(classToBeTested := 0);
	usintAssertions			:UsintAssertionTests(classToBeTested := 0);
	uintAssertions			:UintAssertionTests(classToBeTested := 0);
	udintAssertions			:UdintAssertionTests(classToBeTested := 0);
	ulintAssertions			:UlintAssertionTests(classToBeTested := 0);	
	xintAssertions			:XintAssertionTests(classToBeTested := 0);
	sintAssertions			:SintAssertionTests(classToBeTested := 0);
	intAssertions			:IntAssertionTests(classToBeTested := 0);
	dintAssertions			:DintAssertionTests(classToBeTested := 0);
	lintAssertions			:LintAssertionTests(classToBeTested := 0);
	lrealAssertions		 	:LRealAssertionTests(classToBeTested := 0);
	realAssertions			:RealAssertionTests(classToBeTested := 0);
	bitNumberAssertiosByte	:ByteAssertionTests(classToBeTested := 0);
	bitNumberAssertionsWord :WordAssertionTests(classToBeTested := 0);
	bitNumberAssertionDword	:DWordAssertionTests(classToBeTested := 0);
	bitNumberAssertionLWord :LWordAssertionTests(classToBeTested := 0);
	bitNumberAssertionXWord :XWordAssertionTests(classToBeTested := 0);
	binaryTests				:BinaryAssertionsTests(classToBeTested := 0);
	dateAndTimeAssertions 	:DTAssertionTests(classToBeTested := 0);
	timeTests				:TimeAssertionsTests(classToBeTested := 0);
	stringTests				:StringAssertionTests(classToBeTested := 0);
	objectTests				:ObjectAssertionsTests(classToBeTested := 0);
	dateAssertions			:DateAssertionTests(classToBeTested := 0);
	timeOfDayAssertions 	:TODAssertionTests(classToBeTested := 0);
END_VAR

(*

short summary
=============

.. <legal notes>

legal notes
=================
| SPDX-FileCopyrightText: © 2023 ekvip automation GmbH <info@ekvip.de>
| SPDX-License-Identifier: Apache-2.0
| For details check: Apache-2.0_

.. _Apache-2.0: https://www.apache.org/licenses/LICENSE-2.0

.. </legal notes>

*)

{warning 'header is generated please add your documentation'}
PROPERTY attachAssertorContainer : IAssertorContainer
SET
THIS^.timeTests.attachAssertorContainer					:= attachAssertorContainer;
THIS^.stringTests.attachAssertorContainer 				:= attachAssertorContainer;
THIS^.objectTests.attachAssertorContainer 				:= attachAssertorContainer;
THIS^.pointerTests.attachAssertorContainer 				:= attachAssertorContainer;
THIS^.binaryTests.attachAssertorContainer 				:= attachAssertorContainer;
THIS^.lrealAssertions.attachAssertorContainer 			:= attachAssertorContainer;
THIS^.realAssertions.attachAssertorContainer 			:= attachAssertorContainer;
THIS^.dateAssertions.attachAssertorContainer 			:= attachAssertorContainer;
THIS^.dateAndTimeAssertions.attachAssertorContainer		:= attachAssertorContainer;
THIS^.timeOfDayAssertions.attachAssertorContainer		:= attachAssertorContainer;
THIS^.usintAssertions.attachAssertorContainer			:= attachAssertorContainer;
THIS^.uintAssertions.attachAssertorContainer			:= attachAssertorContainer;
THIS^.udintAssertions.attachAssertorContainer			:= attachAssertorContainer;
THIS^.ulintAssertions.attachAssertorContainer			:= attachAssertorContainer;
THIS^.uxintAssertions.attachAssertorContainer			:= attachAssertorContainer;
THIS^.sintAssertions.attachAssertorContainer			:= attachAssertorContainer;
THIS^.intAssertions.attachAssertorContainer				:= attachAssertorContainer;
THIS^.dintAssertions.attachAssertorContainer			:= attachAssertorContainer;
THIS^.lintAssertions.attachAssertorContainer			:= attachAssertorContainer;
THIS^.xintAssertions.attachAssertorContainer			:= attachAssertorContainer;
THIS^.bitNumberAssertiosByte.attachAssertorContainer	:= attachAssertorContainer;
THIS^.bitNumberAssertionsWord.attachAssertorContainer	:= attachAssertorContainer;
THIS^.bitNumberAssertionDword.attachAssertorContainer	:= attachAssertorContainer;
THIS^.bitNumberAssertionLWord.attachAssertorContainer	:= attachAssertorContainer;
THIS^.bitNumberAssertionXWord.attachAssertorContainer	:= attachAssertorContainer;
END_SET
END_PROPERTY

(*

short summary
=============

.. <legal notes>

legal notes
=================
| SPDX-FileCopyrightText: © 2023 ekvip automation GmbH <info@ekvip.de>
| SPDX-License-Identifier: Apache-2.0
| For details check: Apache-2.0_

.. _Apache-2.0: https://www.apache.org/licenses/LICENSE-2.0

.. </legal notes>

*)

{warning 'header is generated please add your documentation'}
PROPERTY className :CNM_AbstractObject.ClassName
GET
(*

short summary
=============

.. <legal notes>

legal notes
=================
| SPDX-FileCopyrightText: © 2023 ekvip automation GmbH <info@ekvip.de>
| SPDX-License-Identifier: Apache-2.0
| For details check: Apache-2.0_

.. _Apache-2.0: https://www.apache.org/licenses/LICENSE-2.0

.. </legal notes>

*)

{warning 'header is generated please add your documentation'}
VAR
END_VAR
className := 'AssertionTester';
END_GET
END_PROPERTY

(*

short summary
=================
The constructor ``FB_init`` is needed to create an unique hash code.
The hash code is a pseudo random number create with a xorshift_ algorithm.
It can be overwritten on derivations, because it will be called implicit, ``SUPER^.FB_init()`` is not required.
For more information check: `Behavoir with derived function blocks`_

.. _Behavoir with derived function blocks: https://infosys.beckhoff.com/content/1033/tc3_plc_intro/5482088715.html?id=6983869892358031022
.. _xorshift: https://en.wikipedia.org/wiki/Xorshift

.. <legal notes>

legal notes
=================
| SPDX-FileCopyrightText: © 2022 ekvip automation GmbH <info@ekvip.de>
| SPDX-License-Identifier: Apache-2.0
| For details check: Apache-2.0_

.. _Apache-2.0: https://www.apache.org/licenses/LICENSE-2.0

.. </legal notes>

parameters
=================

*)

METHOD FB_init
VAR_INPUT
	(* if TRUE, the retain variables are initialized (warm start / cold start)*)
	bInitRetains	:BOOL;
	(* if TRUE, the instance afterwards gets moved into the copy code (online change) *)
	bInCopyCode		:BOOL;
	(* assertor class to test *)
	classToBeTested :IAssertorContainer;
END_VAR
VAR
	{attribute 'hide'}
	newHashstate3		:Hashcode;
END_VAR
VAR CONSTANT
	{attribute 'hide'}
	NUMBER_OF_LEFT_SHIFTS		:UINT	:= 17;
	{attribute 'hide'}
	NUMBER_OF_LEFT_ROTATIONS	:UINT   := 45;
END_VAR
THIS^.attachAssertorContainer := classToBeTested;
END_METHOD

END_FUNCTION_BLOCK

// ---- AssertionTester/functions/ArrayOfMessageStringToString.TcPOU
(*

short summary
=============

.. <legal notes>

legal notes
=================
| SPDX-FileCopyrightText: © 2023 ekvip automation GmbH <info@ekvip.de>
| SPDX-License-Identifier: Apache-2.0
| For details check: Apache-2.0_

.. _Apache-2.0: https://www.apache.org/licenses/LICENSE-2.0

.. </legal notes>

parameters
==========

*)

{warning 'header is generated please add your documentation'}
FUNCTION ArrayOfMessageStringToString : Tc2_System.T_MaxString
VAR_IN_OUT
	message :ARRAY [*] OF STRING;
END_VAR
VAR
	i :INT := 0;
	tempString :STRING := '';
END_VAR

WHILE (message[i] <> '#END') DO
	tempString := CONCAT(tempString, message[i]);
	i:= i + 1;
	IF (i >= 10) THEN
		EXIT;
	END_IF
END_WHILE

ArrayOfMessageStringToString := tempString;

END_FUNCTION

// ---- Project Information/F_GetCompany.TcPOU
// This function has been automatically generated from the project information.
{attribute 'signature_flag' := '1073741824'}
{attribute 'TcGenerated'}
{attribute 'no-analysis'}
FUNCTION F_GetCompany : WSTRING
VAR_INPUT
	
END_VAR

F_GetCompany := "ekvip automation GmbH";

END_FUNCTION

// ---- Project Information/F_GetTitle.TcPOU
// This function has been automatically generated from the project information.
{attribute 'signature_flag' := '1073741824'}
{attribute 'TcGenerated'}
{attribute 'no-analysis'}
FUNCTION F_GetTitle : WSTRING
VAR_INPUT
	
END_VAR

F_GetTitle := "CNM_AssertionInterfaceTests";

END_FUNCTION

// ---- Project Information/F_GetVersion.TcPOU
// This function has been automatically generated from the project information.
{attribute 'signature_flag' := '1073741824'}
{attribute 'TcGenerated'}
{attribute 'no-analysis'}
FUNCTION F_GetVersion : ST_LibVersion
VAR_INPUT
	
END_VAR

F_GetVersion.iMajor := 1;
F_GetVersion.iMinor := 0;
F_GetVersion.iBuild := 0;
F_GetVersion.iRevision := 47;
F_GetVersion.sVersion := '1.0.0.47';
F_GetVersion.nFlags := 0;

END_FUNCTION
